REGION Network 36: UNIT 1 STATION 3 MEASURING RESET METHOD CONNECTION ALARM
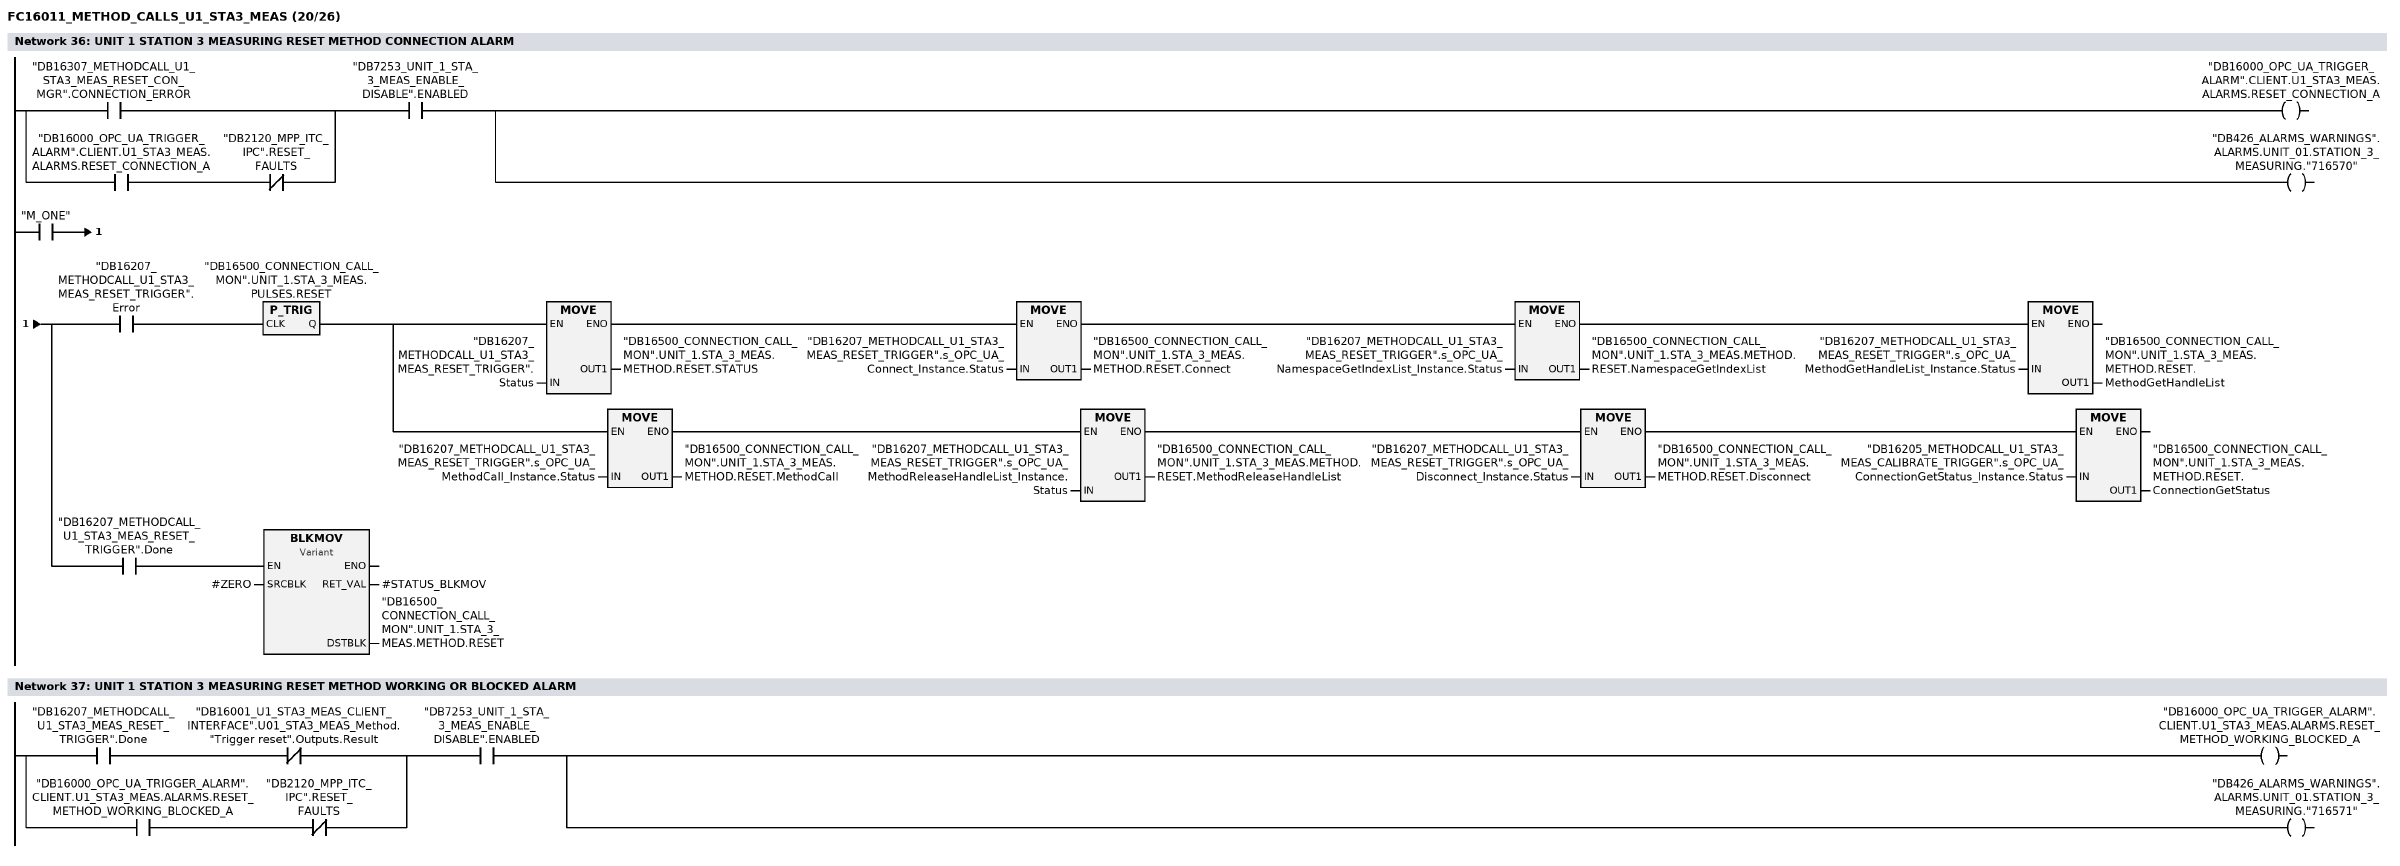
   RUNG wire#powerrail
      Contact( "DB16307_METHODCALL_U1_STA3_MEAS_RESET_CON_MGR".CONNECTION_ERROR )
      wire#w1
      Contact( "DB7253_UNIT_1_STA_3_MEAS_ENABLE_DISABLE".ENABLED )
      wire#w2
      Coil( "DB16000_OPC_UA_TRIGGER_ALARM".CLIENT.U1_STA3_MEAS.ALARMS.RESET_CONNECTION_A )
   END_RUNG
   RUNG wire#powerrail
      Contact( "DB16000_OPC_UA_TRIGGER_ALARM".CLIENT.U1_STA3_MEAS.ALARMS.RESET_CONNECTION_A )
      I_Contact( "DB2120_MPP_ITC_IPC".RESET_FAULTS )
   END_RUNG wire#w1
   RUNG wire#w2
      Coil( "DB426_ALARMS_WARNINGS".ALARMS.UNIT_01.STATION_3_MEASURING."716570" )
   END_RUNG
   RUNG wire#powerrail
      Contact( "M_ONE" )
      wire#w3
      Contact( "DB16207_METHODCALL_U1_STA3_MEAS_RESET_TRIGGER".Error )
      P_Trig( "DB16500_CONNECTION_CALL_MON".UNIT_1.STA_3_MEAS.PULSES.RESET )
      wire#w4
      Move(in := "DB16207_METHODCALL_U1_STA3_MEAS_RESET_TRIGGER".Status, out1 => "DB16500_CONNECTION_CALL_MON".UNIT_1.STA_3_MEAS.METHOD.RESET.STATUS)
      Move(in := "DB16207_METHODCALL_U1_STA3_MEAS_RESET_TRIGGER".s_OPC_UA_Connect_Instance.Status, out1 => "DB16500_CONNECTION_CALL_MON".UNIT_1.STA_3_MEAS.METHOD.RESET.Connect)
      Move(in := "DB16207_METHODCALL_U1_STA3_MEAS_RESET_TRIGGER".s_OPC_UA_NamespaceGetIndexList_Instance.Status, out1 => "DB16500_CONNECTION_CALL_MON".UNIT_1.STA_3_MEAS.METHOD.RESET.NamespaceGetIndexList)
      Move(in := "DB16207_METHODCALL_U1_STA3_MEAS_RESET_TRIGGER".s_OPC_UA_MethodGetHandleList_Instance.Status, out1 => "DB16500_CONNECTION_CALL_MON".UNIT_1.STA_3_MEAS.METHOD.RESET.MethodGetHandleList)
   END_RUNG
   RUNG wire#w4
      Move(in := "DB16207_METHODCALL_U1_STA3_MEAS_RESET_TRIGGER".s_OPC_UA_MethodCall_Instance.Status, out1 => "DB16500_CONNECTION_CALL_MON".UNIT_1.STA_3_MEAS.METHOD.RESET.MethodCall)
      Move(in := "DB16207_METHODCALL_U1_STA3_MEAS_RESET_TRIGGER".s_OPC_UA_MethodReleaseHandleList_Instance.Status, out1 => "DB16500_CONNECTION_CALL_MON".UNIT_1.STA_3_MEAS.METHOD.RESET.MethodReleaseHandleList)
      Move(in := "DB16207_METHODCALL_U1_STA3_MEAS_RESET_TRIGGER".s_OPC_UA_Disconnect_Instance.Status, out1 => "DB16500_CONNECTION_CALL_MON".UNIT_1.STA_3_MEAS.METHOD.RESET.Disconnect)
      Move(in := "DB16205_METHODCALL_U1_STA3_MEAS_CALIBRATE_TRIGGER".s_OPC_UA_ConnectionGetStatus_Instance.Status, out1 => "DB16500_CONNECTION_CALL_MON".UNIT_1.STA_3_MEAS.METHOD.RESET.ConnectionGetStatus)
   END_RUNG
   RUNG wire#w3
      Contact( "DB16207_METHODCALL_U1_STA3_MEAS_RESET_TRIGGER".Done )
      { S7_Templates := "blk_type := Variant" } BLKMOV(SRCBLK := #ZERO, RET_VAL => #STATUS_BLKMOV, DSTBLK => "DB16500_CONNECTION_CALL_MON".UNIT_1.STA_3_MEAS.METHOD.RESET)
   END_RUNG
   // the same network as SCL:
   "DB16000_OPC_UA_TRIGGER_ALARM".CLIENT.U1_STA3_MEAS.ALARMS.RESET_CONNECTION_A := ("DB16307_METHODCALL_U1_STA3_MEAS_RESET_CON_MGR".CONNECTION_ERROR OR ("DB16000_OPC_UA_TRIGGER_ALARM".CLIENT.U1_STA3_MEAS.ALARMS.RESET_CONNECTION_A AND NOT "DB2120_MPP_ITC_IPC".RESET_FAULTS)) AND "DB7253_UNIT_1_STA_3_MEAS_ENABLE_DISABLE".ENABLED;
   "DB426_ALARMS_WARNINGS".ALARMS.UNIT_01.STATION_3_MEASURING."716570" := "DB16000_OPC_UA_TRIGGER_ALARM".CLIENT.U1_STA3_MEAS.ALARMS.RESET_CONNECTION_A;
   #_w1 := "M_ONE" AND "DB16207_METHODCALL_U1_STA3_MEAS_RESET_TRIGGER".Error;
   #_w2 := #_w1 AND NOT "DB16500_CONNECTION_CALL_MON".UNIT_1.STA_3_MEAS.PULSES.RESET;   // rising edge
   "DB16500_CONNECTION_CALL_MON".UNIT_1.STA_3_MEAS.PULSES.RESET := #_w1;
   IF #_w2 THEN
       "DB16500_CONNECTION_CALL_MON".UNIT_1.STA_3_MEAS.METHOD.RESET.STATUS := "DB16207_METHODCALL_U1_STA3_MEAS_RESET_TRIGGER".Status;
       "DB16500_CONNECTION_CALL_MON".UNIT_1.STA_3_MEAS.METHOD.RESET.Connect := "DB16207_METHODCALL_U1_STA3_MEAS_RESET_TRIGGER".s_OPC_UA_Connect_Instance.Status;
       "DB16500_CONNECTION_CALL_MON".UNIT_1.STA_3_MEAS.METHOD.RESET.NamespaceGetIndexList := "DB16207_METHODCALL_U1_STA3_MEAS_RESET_TRIGGER".s_OPC_UA_NamespaceGetIndexList_Instance.Status;
       "DB16500_CONNECTION_CALL_MON".UNIT_1.STA_3_MEAS.METHOD.RESET.MethodGetHandleList := "DB16207_METHODCALL_U1_STA3_MEAS_RESET_TRIGGER".s_OPC_UA_MethodGetHandleList_Instance.Status;
       "DB16500_CONNECTION_CALL_MON".UNIT_1.STA_3_MEAS.METHOD.RESET.MethodCall := "DB16207_METHODCALL_U1_STA3_MEAS_RESET_TRIGGER".s_OPC_UA_MethodCall_Instance.Status;
       "DB16500_CONNECTION_CALL_MON".UNIT_1.STA_3_MEAS.METHOD.RESET.MethodReleaseHandleList := "DB16207_METHODCALL_U1_STA3_MEAS_RESET_TRIGGER".s_OPC_UA_MethodReleaseHandleList_Instance.Status;
       "DB16500_CONNECTION_CALL_MON".UNIT_1.STA_3_MEAS.METHOD.RESET.Disconnect := "DB16207_METHODCALL_U1_STA3_MEAS_RESET_TRIGGER".s_OPC_UA_Disconnect_Instance.Status;
       "DB16500_CONNECTION_CALL_MON".UNIT_1.STA_3_MEAS.METHOD.RESET.ConnectionGetStatus := "DB16205_METHODCALL_U1_STA3_MEAS_CALIBRATE_TRIGGER".s_OPC_UA_ConnectionGetStatus_Instance.Status;
   END_IF;
   IF "M_ONE" AND "DB16207_METHODCALL_U1_STA3_MEAS_RESET_TRIGGER".Done THEN
       #STATUS_BLKMOV := BLKMOV(SRCBLK := #ZERO,
                               DSTBLK => "DB16500_CONNECTION_CALL_MON".UNIT_1.STA_3_MEAS.METHOD.RESET);
   END_IF;
END_REGION

REGION Network 37: UNIT 1 STATION 3 MEASURING RESET METHOD WORKING OR BLOCKED ALARM
   RUNG wire#powerrail
      Contact( "DB16207_METHODCALL_U1_STA3_MEAS_RESET_TRIGGER".Done )
      I_Contact( "DB16001_U1_STA3_MEAS_CLIENT_INTERFACE".U01_STA3_MEAS_Method."Trigger reset".Outputs.Result )
      wire#w1
      Contact( "DB7253_UNIT_1_STA_3_MEAS_ENABLE_DISABLE".ENABLED )
      wire#w2
      Coil( "DB16000_OPC_UA_TRIGGER_ALARM".CLIENT.U1_STA3_MEAS.ALARMS.RESET_METHOD_WORKING_BLOCKED_A )
   END_RUNG
   RUNG wire#powerrail
      Contact( "DB16000_OPC_UA_TRIGGER_ALARM".CLIENT.U1_STA3_MEAS.ALARMS.RESET_METHOD_WORKING_BLOCKED_A )
      I_Contact( "DB2120_MPP_ITC_IPC".RESET_FAULTS )
   END_RUNG wire#w1
   RUNG wire#w2
      Coil( "DB426_ALARMS_WARNINGS".ALARMS.UNIT_01.STATION_3_MEASURING."716571" )
   END_RUNG
   // the same network as SCL:
   "DB16000_OPC_UA_TRIGGER_ALARM".CLIENT.U1_STA3_MEAS.ALARMS.RESET_METHOD_WORKING_BLOCKED_A := (("DB16207_METHODCALL_U1_STA3_MEAS_RESET_TRIGGER".Done AND NOT "DB16001_U1_STA3_MEAS_CLIENT_INTERFACE".U01_STA3_MEAS_Method."Trigger reset".Outputs.Result) OR ("DB16000_OPC_UA_TRIGGER_ALARM".CLIENT.U1_STA3_MEAS.ALARMS.RESET_METHOD_WORKING_BLOCKED_A AND NOT "DB2120_MPP_ITC_IPC".RESET_FAULTS)) AND "DB7253_UNIT_1_STA_3_MEAS_ENABLE_DISABLE".ENABLED;
   "DB426_ALARMS_WARNINGS".ALARMS.UNIT_01.STATION_3_MEASURING."716571" := "DB16000_OPC_UA_TRIGGER_ALARM".CLIENT.U1_STA3_MEAS.ALARMS.RESET_METHOD_WORKING_BLOCKED_A;
END_REGION

REGION Network 38: UNIT 1 STATION 3 MEASURING READ VARIABLES CONNECTION ALARM
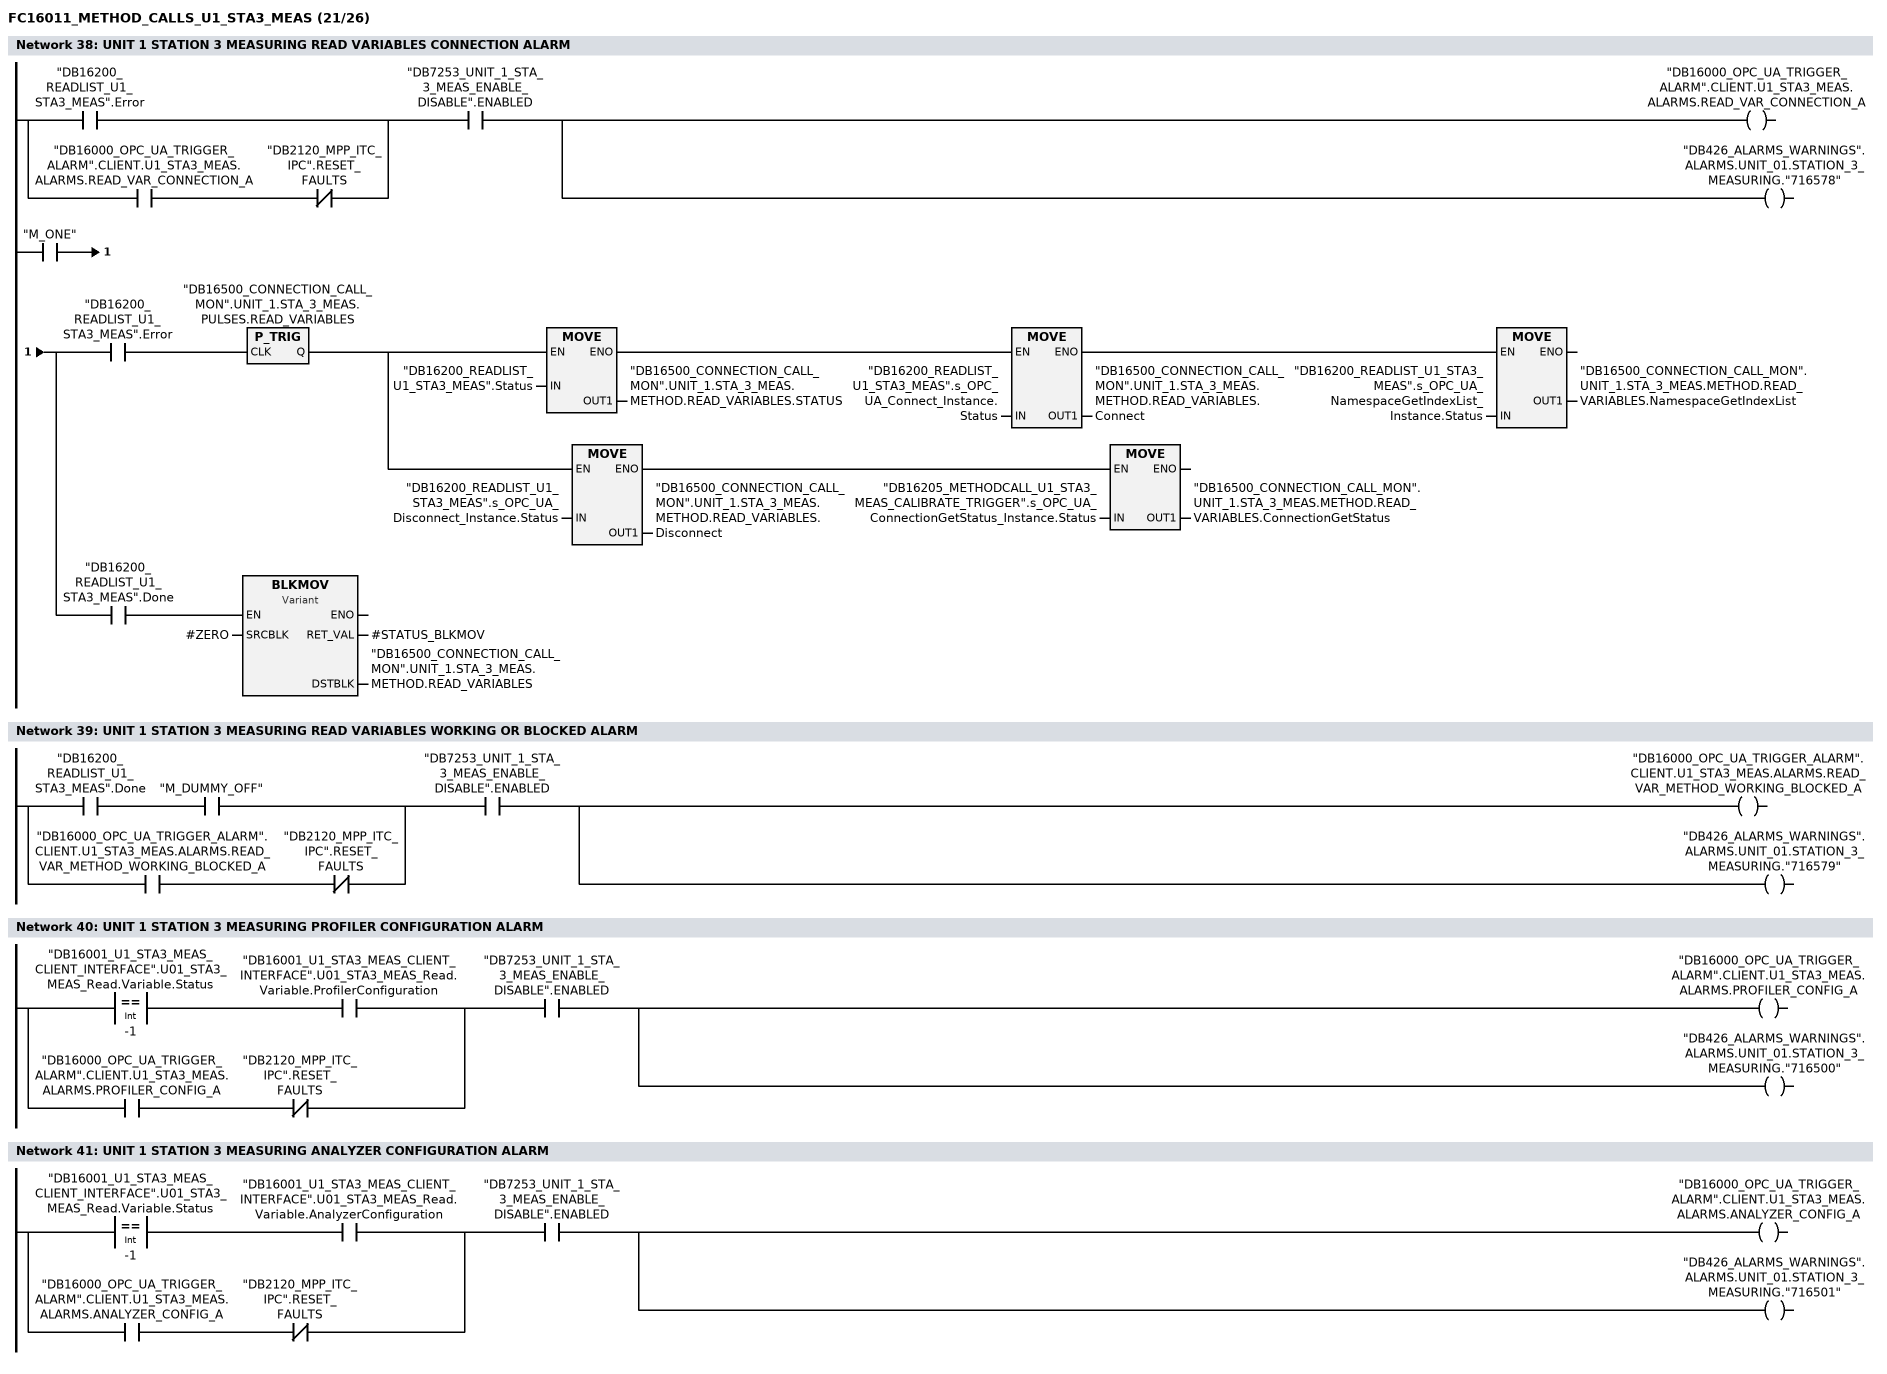
   RUNG wire#powerrail
      Contact( "DB16200_READLIST_U1_STA3_MEAS".Error )
      wire#w1
      Contact( "DB7253_UNIT_1_STA_3_MEAS_ENABLE_DISABLE".ENABLED )
      wire#w2
      Coil( "DB16000_OPC_UA_TRIGGER_ALARM".CLIENT.U1_STA3_MEAS.ALARMS.READ_VAR_CONNECTION_A )
   END_RUNG
   RUNG wire#powerrail
      Contact( "DB16000_OPC_UA_TRIGGER_ALARM".CLIENT.U1_STA3_MEAS.ALARMS.READ_VAR_CONNECTION_A )
      I_Contact( "DB2120_MPP_ITC_IPC".RESET_FAULTS )
   END_RUNG wire#w1
   RUNG wire#w2
      Coil( "DB426_ALARMS_WARNINGS".ALARMS.UNIT_01.STATION_3_MEASURING."716578" )
   END_RUNG
   RUNG wire#powerrail
      Contact( "M_ONE" )
      wire#w3
      Contact( "DB16200_READLIST_U1_STA3_MEAS".Error )
      P_Trig( "DB16500_CONNECTION_CALL_MON".UNIT_1.STA_3_MEAS.PULSES.READ_VARIABLES )
      wire#w4
      Move(in := "DB16200_READLIST_U1_STA3_MEAS".Status, out1 => "DB16500_CONNECTION_CALL_MON".UNIT_1.STA_3_MEAS.METHOD.READ_VARIABLES.STATUS)
      Move(in := "DB16200_READLIST_U1_STA3_MEAS".s_OPC_UA_Connect_Instance.Status, out1 => "DB16500_CONNECTION_CALL_MON".UNIT_1.STA_3_MEAS.METHOD.READ_VARIABLES.Connect)
      Move(in := "DB16200_READLIST_U1_STA3_MEAS".s_OPC_UA_NamespaceGetIndexList_Instance.Status, out1 => "DB16500_CONNECTION_CALL_MON".UNIT_1.STA_3_MEAS.METHOD.READ_VARIABLES.NamespaceGetIndexList)
   END_RUNG
   RUNG wire#w4
      Move(in := "DB16200_READLIST_U1_STA3_MEAS".s_OPC_UA_Disconnect_Instance.Status, out1 => "DB16500_CONNECTION_CALL_MON".UNIT_1.STA_3_MEAS.METHOD.READ_VARIABLES.Disconnect)
      Move(in := "DB16205_METHODCALL_U1_STA3_MEAS_CALIBRATE_TRIGGER".s_OPC_UA_ConnectionGetStatus_Instance.Status, out1 => "DB16500_CONNECTION_CALL_MON".UNIT_1.STA_3_MEAS.METHOD.READ_VARIABLES.ConnectionGetStatus)
   END_RUNG
   RUNG wire#w3
      Contact( "DB16200_READLIST_U1_STA3_MEAS".Done )
      { S7_Templates := "blk_type := Variant" } BLKMOV(SRCBLK := #ZERO, RET_VAL => #STATUS_BLKMOV, DSTBLK => "DB16500_CONNECTION_CALL_MON".UNIT_1.STA_3_MEAS.METHOD.READ_VARIABLES)
   END_RUNG
   // the same network as SCL:
   "DB16000_OPC_UA_TRIGGER_ALARM".CLIENT.U1_STA3_MEAS.ALARMS.READ_VAR_CONNECTION_A := ("DB16200_READLIST_U1_STA3_MEAS".Error OR ("DB16000_OPC_UA_TRIGGER_ALARM".CLIENT.U1_STA3_MEAS.ALARMS.READ_VAR_CONNECTION_A AND NOT "DB2120_MPP_ITC_IPC".RESET_FAULTS)) AND "DB7253_UNIT_1_STA_3_MEAS_ENABLE_DISABLE".ENABLED;
   "DB426_ALARMS_WARNINGS".ALARMS.UNIT_01.STATION_3_MEASURING."716578" := "DB16000_OPC_UA_TRIGGER_ALARM".CLIENT.U1_STA3_MEAS.ALARMS.READ_VAR_CONNECTION_A;
   #_w1 := "M_ONE" AND "DB16200_READLIST_U1_STA3_MEAS".Error;
   #_w2 := #_w1 AND NOT "DB16500_CONNECTION_CALL_MON".UNIT_1.STA_3_MEAS.PULSES.READ_VARIABLES;   // rising edge
   "DB16500_CONNECTION_CALL_MON".UNIT_1.STA_3_MEAS.PULSES.READ_VARIABLES := #_w1;
   IF #_w2 THEN
       "DB16500_CONNECTION_CALL_MON".UNIT_1.STA_3_MEAS.METHOD.READ_VARIABLES.STATUS := "DB16200_READLIST_U1_STA3_MEAS".Status;
       "DB16500_CONNECTION_CALL_MON".UNIT_1.STA_3_MEAS.METHOD.READ_VARIABLES.Connect := "DB16200_READLIST_U1_STA3_MEAS".s_OPC_UA_Connect_Instance.Status;
       "DB16500_CONNECTION_CALL_MON".UNIT_1.STA_3_MEAS.METHOD.READ_VARIABLES.NamespaceGetIndexList := "DB16200_READLIST_U1_STA3_MEAS".s_OPC_UA_NamespaceGetIndexList_Instance.Status;
       "DB16500_CONNECTION_CALL_MON".UNIT_1.STA_3_MEAS.METHOD.READ_VARIABLES.Disconnect := "DB16200_READLIST_U1_STA3_MEAS".s_OPC_UA_Disconnect_Instance.Status;
       "DB16500_CONNECTION_CALL_MON".UNIT_1.STA_3_MEAS.METHOD.READ_VARIABLES.ConnectionGetStatus := "DB16205_METHODCALL_U1_STA3_MEAS_CALIBRATE_TRIGGER".s_OPC_UA_ConnectionGetStatus_Instance.Status;
   END_IF;
   IF "M_ONE" AND "DB16200_READLIST_U1_STA3_MEAS".Done THEN
       #STATUS_BLKMOV := BLKMOV(SRCBLK := #ZERO,
                               DSTBLK => "DB16500_CONNECTION_CALL_MON".UNIT_1.STA_3_MEAS.METHOD.READ_VARIABLES);
   END_IF;
END_REGION

REGION Network 39: UNIT 1 STATION 3 MEASURING READ VARIABLES WORKING OR BLOCKED ALARM
   RUNG wire#powerrail
      Contact( "DB16200_READLIST_U1_STA3_MEAS".Done )
      Contact( "M_DUMMY_OFF" )
      wire#w1
      Contact( "DB7253_UNIT_1_STA_3_MEAS_ENABLE_DISABLE".ENABLED )
      wire#w2
      Coil( "DB16000_OPC_UA_TRIGGER_ALARM".CLIENT.U1_STA3_MEAS.ALARMS.READ_VAR_METHOD_WORKING_BLOCKED_A )
   END_RUNG
   RUNG wire#powerrail
      Contact( "DB16000_OPC_UA_TRIGGER_ALARM".CLIENT.U1_STA3_MEAS.ALARMS.READ_VAR_METHOD_WORKING_BLOCKED_A )
      I_Contact( "DB2120_MPP_ITC_IPC".RESET_FAULTS )
   END_RUNG wire#w1
   RUNG wire#w2
      Coil( "DB426_ALARMS_WARNINGS".ALARMS.UNIT_01.STATION_3_MEASURING."716579" )
   END_RUNG
   // the same network as SCL:
   "DB16000_OPC_UA_TRIGGER_ALARM".CLIENT.U1_STA3_MEAS.ALARMS.READ_VAR_METHOD_WORKING_BLOCKED_A := (("DB16200_READLIST_U1_STA3_MEAS".Done AND "M_DUMMY_OFF") OR ("DB16000_OPC_UA_TRIGGER_ALARM".CLIENT.U1_STA3_MEAS.ALARMS.READ_VAR_METHOD_WORKING_BLOCKED_A AND NOT "DB2120_MPP_ITC_IPC".RESET_FAULTS)) AND "DB7253_UNIT_1_STA_3_MEAS_ENABLE_DISABLE".ENABLED;
   "DB426_ALARMS_WARNINGS".ALARMS.UNIT_01.STATION_3_MEASURING."716579" := "DB16000_OPC_UA_TRIGGER_ALARM".CLIENT.U1_STA3_MEAS.ALARMS.READ_VAR_METHOD_WORKING_BLOCKED_A;
END_REGION

REGION Network 40: UNIT 1 STATION 3 MEASURING PROFILER CONFIGURATION ALARM
   RUNG wire#powerrail
      { S7_Templates := "SrcType := Int" } EQ_Contact(in1 := "DB16001_U1_STA3_MEAS_CLIENT_INTERFACE".U01_STA3_MEAS_Read.Variable.Status, in2 := -1)
      Contact( "DB16001_U1_STA3_MEAS_CLIENT_INTERFACE".U01_STA3_MEAS_Read.Variable.ProfilerConfiguration )
      wire#w1
      Contact( "DB7253_UNIT_1_STA_3_MEAS_ENABLE_DISABLE".ENABLED )
      wire#w2
      Coil( "DB16000_OPC_UA_TRIGGER_ALARM".CLIENT.U1_STA3_MEAS.ALARMS.PROFILER_CONFIG_A )
   END_RUNG
   RUNG wire#powerrail
      Contact( "DB16000_OPC_UA_TRIGGER_ALARM".CLIENT.U1_STA3_MEAS.ALARMS.PROFILER_CONFIG_A )
      I_Contact( "DB2120_MPP_ITC_IPC".RESET_FAULTS )
   END_RUNG wire#w1
   RUNG wire#w2
      Coil( "DB426_ALARMS_WARNINGS".ALARMS.UNIT_01.STATION_3_MEASURING."716500" )
   END_RUNG
   // the same network as SCL:
   "DB16000_OPC_UA_TRIGGER_ALARM".CLIENT.U1_STA3_MEAS.ALARMS.PROFILER_CONFIG_A := ((("DB16001_U1_STA3_MEAS_CLIENT_INTERFACE".U01_STA3_MEAS_Read.Variable.Status = (-1)) AND "DB16001_U1_STA3_MEAS_CLIENT_INTERFACE".U01_STA3_MEAS_Read.Variable.ProfilerConfiguration) OR ("DB16000_OPC_UA_TRIGGER_ALARM".CLIENT.U1_STA3_MEAS.ALARMS.PROFILER_CONFIG_A AND NOT "DB2120_MPP_ITC_IPC".RESET_FAULTS)) AND "DB7253_UNIT_1_STA_3_MEAS_ENABLE_DISABLE".ENABLED;
   "DB426_ALARMS_WARNINGS".ALARMS.UNIT_01.STATION_3_MEASURING."716500" := "DB16000_OPC_UA_TRIGGER_ALARM".CLIENT.U1_STA3_MEAS.ALARMS.PROFILER_CONFIG_A;
END_REGION

REGION Network 41: UNIT 1 STATION 3 MEASURING ANALYZER CONFIGURATION ALARM
   RUNG wire#powerrail
      { S7_Templates := "SrcType := Int" } EQ_Contact(in1 := "DB16001_U1_STA3_MEAS_CLIENT_INTERFACE".U01_STA3_MEAS_Read.Variable.Status, in2 := -1)
      Contact( "DB16001_U1_STA3_MEAS_CLIENT_INTERFACE".U01_STA3_MEAS_Read.Variable.AnalyzerConfiguration )
      wire#w1
      Contact( "DB7253_UNIT_1_STA_3_MEAS_ENABLE_DISABLE".ENABLED )
      wire#w2
      Coil( "DB16000_OPC_UA_TRIGGER_ALARM".CLIENT.U1_STA3_MEAS.ALARMS.ANALYZER_CONFIG_A )
   END_RUNG
   RUNG wire#powerrail
      Contact( "DB16000_OPC_UA_TRIGGER_ALARM".CLIENT.U1_STA3_MEAS.ALARMS.ANALYZER_CONFIG_A )
      I_Contact( "DB2120_MPP_ITC_IPC".RESET_FAULTS )
   END_RUNG wire#w1
   RUNG wire#w2
      Coil( "DB426_ALARMS_WARNINGS".ALARMS.UNIT_01.STATION_3_MEASURING."716501" )
   END_RUNG
   // the same network as SCL:
   "DB16000_OPC_UA_TRIGGER_ALARM".CLIENT.U1_STA3_MEAS.ALARMS.ANALYZER_CONFIG_A := ((("DB16001_U1_STA3_MEAS_CLIENT_INTERFACE".U01_STA3_MEAS_Read.Variable.Status = (-1)) AND "DB16001_U1_STA3_MEAS_CLIENT_INTERFACE".U01_STA3_MEAS_Read.Variable.AnalyzerConfiguration) OR ("DB16000_OPC_UA_TRIGGER_ALARM".CLIENT.U1_STA3_MEAS.ALARMS.ANALYZER_CONFIG_A AND NOT "DB2120_MPP_ITC_IPC".RESET_FAULTS)) AND "DB7253_UNIT_1_STA_3_MEAS_ENABLE_DISABLE".ENABLED;
   "DB426_ALARMS_WARNINGS".ALARMS.UNIT_01.STATION_3_MEASURING."716501" := "DB16000_OPC_UA_TRIGGER_ALARM".CLIENT.U1_STA3_MEAS.ALARMS.ANALYZER_CONFIG_A;
END_REGION

REGION Network 42: UNIT 1 STATION 3 MEASURING DMC STRUCTURE ALARM
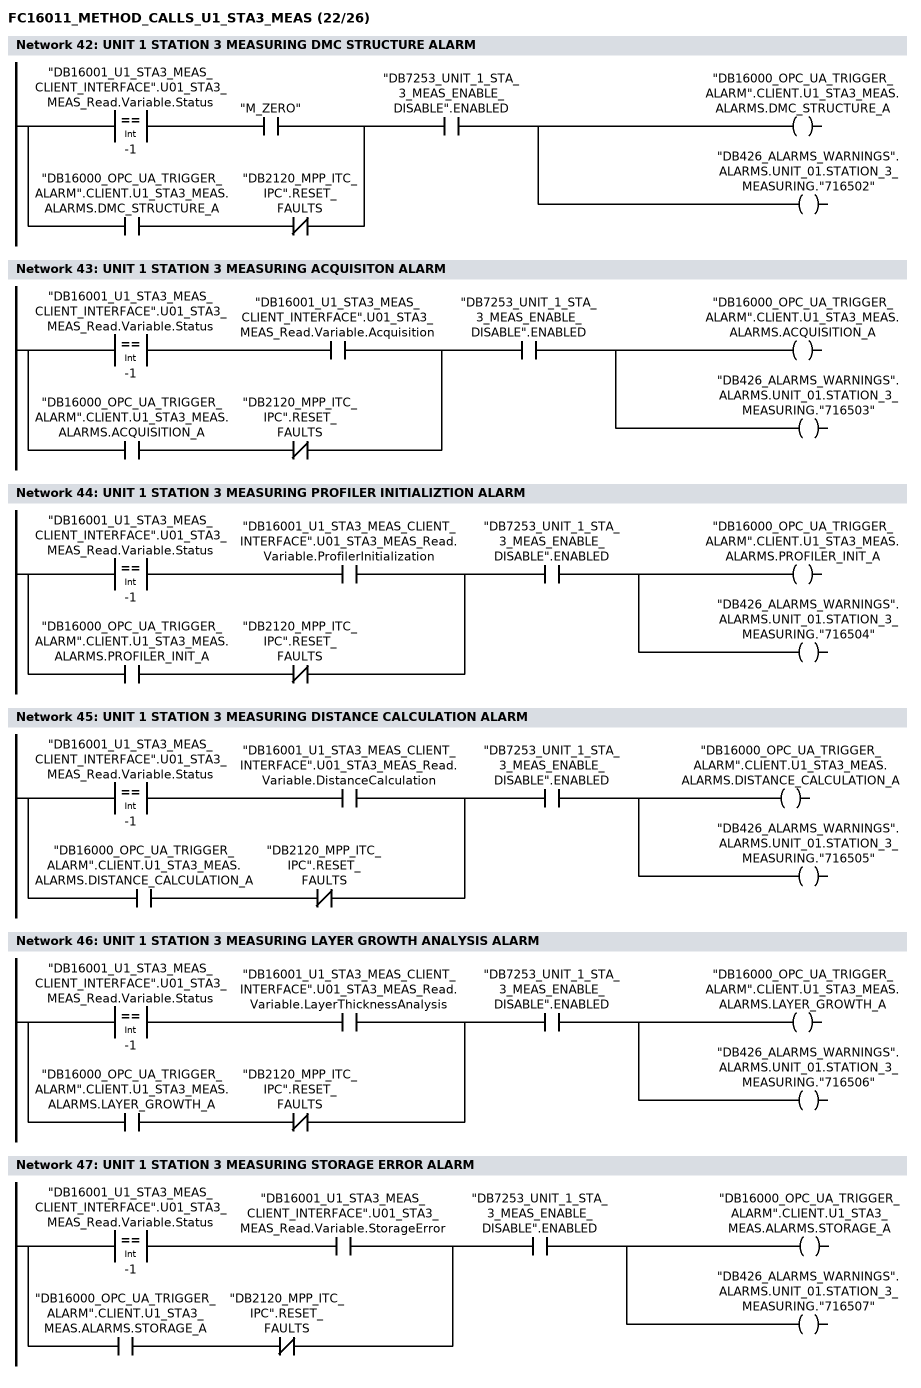
   RUNG wire#powerrail
      { S7_Templates := "SrcType := Int" } EQ_Contact(in1 := "DB16001_U1_STA3_MEAS_CLIENT_INTERFACE".U01_STA3_MEAS_Read.Variable.Status, in2 := -1)
      Contact( "M_ZERO" )
      wire#w1
      Contact( "DB7253_UNIT_1_STA_3_MEAS_ENABLE_DISABLE".ENABLED )
      wire#w2
      Coil( "DB16000_OPC_UA_TRIGGER_ALARM".CLIENT.U1_STA3_MEAS.ALARMS.DMC_STRUCTURE_A )
   END_RUNG
   RUNG wire#powerrail
      Contact( "DB16000_OPC_UA_TRIGGER_ALARM".CLIENT.U1_STA3_MEAS.ALARMS.DMC_STRUCTURE_A )
      I_Contact( "DB2120_MPP_ITC_IPC".RESET_FAULTS )
   END_RUNG wire#w1
   RUNG wire#w2
      Coil( "DB426_ALARMS_WARNINGS".ALARMS.UNIT_01.STATION_3_MEASURING."716502" )
   END_RUNG
   // the same network as SCL:
   "DB16000_OPC_UA_TRIGGER_ALARM".CLIENT.U1_STA3_MEAS.ALARMS.DMC_STRUCTURE_A := ((("DB16001_U1_STA3_MEAS_CLIENT_INTERFACE".U01_STA3_MEAS_Read.Variable.Status = (-1)) AND "M_ZERO") OR ("DB16000_OPC_UA_TRIGGER_ALARM".CLIENT.U1_STA3_MEAS.ALARMS.DMC_STRUCTURE_A AND NOT "DB2120_MPP_ITC_IPC".RESET_FAULTS)) AND "DB7253_UNIT_1_STA_3_MEAS_ENABLE_DISABLE".ENABLED;
   "DB426_ALARMS_WARNINGS".ALARMS.UNIT_01.STATION_3_MEASURING."716502" := "DB16000_OPC_UA_TRIGGER_ALARM".CLIENT.U1_STA3_MEAS.ALARMS.DMC_STRUCTURE_A;
END_REGION

REGION Network 43: UNIT 1 STATION 3 MEASURING ACQUISITON ALARM
   RUNG wire#powerrail
      { S7_Templates := "SrcType := Int" } EQ_Contact(in1 := "DB16001_U1_STA3_MEAS_CLIENT_INTERFACE".U01_STA3_MEAS_Read.Variable.Status, in2 := -1)
      Contact( "DB16001_U1_STA3_MEAS_CLIENT_INTERFACE".U01_STA3_MEAS_Read.Variable.Acquisition )
      wire#w1
      Contact( "DB7253_UNIT_1_STA_3_MEAS_ENABLE_DISABLE".ENABLED )
      wire#w2
      Coil( "DB16000_OPC_UA_TRIGGER_ALARM".CLIENT.U1_STA3_MEAS.ALARMS.ACQUISITION_A )
   END_RUNG
   RUNG wire#powerrail
      Contact( "DB16000_OPC_UA_TRIGGER_ALARM".CLIENT.U1_STA3_MEAS.ALARMS.ACQUISITION_A )
      I_Contact( "DB2120_MPP_ITC_IPC".RESET_FAULTS )
   END_RUNG wire#w1
   RUNG wire#w2
      Coil( "DB426_ALARMS_WARNINGS".ALARMS.UNIT_01.STATION_3_MEASURING."716503" )
   END_RUNG
   // the same network as SCL:
   "DB16000_OPC_UA_TRIGGER_ALARM".CLIENT.U1_STA3_MEAS.ALARMS.ACQUISITION_A := ((("DB16001_U1_STA3_MEAS_CLIENT_INTERFACE".U01_STA3_MEAS_Read.Variable.Status = (-1)) AND "DB16001_U1_STA3_MEAS_CLIENT_INTERFACE".U01_STA3_MEAS_Read.Variable.Acquisition) OR ("DB16000_OPC_UA_TRIGGER_ALARM".CLIENT.U1_STA3_MEAS.ALARMS.ACQUISITION_A AND NOT "DB2120_MPP_ITC_IPC".RESET_FAULTS)) AND "DB7253_UNIT_1_STA_3_MEAS_ENABLE_DISABLE".ENABLED;
   "DB426_ALARMS_WARNINGS".ALARMS.UNIT_01.STATION_3_MEASURING."716503" := "DB16000_OPC_UA_TRIGGER_ALARM".CLIENT.U1_STA3_MEAS.ALARMS.ACQUISITION_A;
END_REGION

REGION Network 44: UNIT 1 STATION 3 MEASURING PROFILER INITIALIZTION ALARM
   RUNG wire#powerrail
      { S7_Templates := "SrcType := Int" } EQ_Contact(in1 := "DB16001_U1_STA3_MEAS_CLIENT_INTERFACE".U01_STA3_MEAS_Read.Variable.Status, in2 := -1)
      Contact( "DB16001_U1_STA3_MEAS_CLIENT_INTERFACE".U01_STA3_MEAS_Read.Variable.ProfilerInitialization )
      wire#w1
      Contact( "DB7253_UNIT_1_STA_3_MEAS_ENABLE_DISABLE".ENABLED )
      wire#w2
      Coil( "DB16000_OPC_UA_TRIGGER_ALARM".CLIENT.U1_STA3_MEAS.ALARMS.PROFILER_INIT_A )
   END_RUNG
   RUNG wire#powerrail
      Contact( "DB16000_OPC_UA_TRIGGER_ALARM".CLIENT.U1_STA3_MEAS.ALARMS.PROFILER_INIT_A )
      I_Contact( "DB2120_MPP_ITC_IPC".RESET_FAULTS )
   END_RUNG wire#w1
   RUNG wire#w2
      Coil( "DB426_ALARMS_WARNINGS".ALARMS.UNIT_01.STATION_3_MEASURING."716504" )
   END_RUNG
   // the same network as SCL:
   "DB16000_OPC_UA_TRIGGER_ALARM".CLIENT.U1_STA3_MEAS.ALARMS.PROFILER_INIT_A := ((("DB16001_U1_STA3_MEAS_CLIENT_INTERFACE".U01_STA3_MEAS_Read.Variable.Status = (-1)) AND "DB16001_U1_STA3_MEAS_CLIENT_INTERFACE".U01_STA3_MEAS_Read.Variable.ProfilerInitialization) OR ("DB16000_OPC_UA_TRIGGER_ALARM".CLIENT.U1_STA3_MEAS.ALARMS.PROFILER_INIT_A AND NOT "DB2120_MPP_ITC_IPC".RESET_FAULTS)) AND "DB7253_UNIT_1_STA_3_MEAS_ENABLE_DISABLE".ENABLED;
   "DB426_ALARMS_WARNINGS".ALARMS.UNIT_01.STATION_3_MEASURING."716504" := "DB16000_OPC_UA_TRIGGER_ALARM".CLIENT.U1_STA3_MEAS.ALARMS.PROFILER_INIT_A;
END_REGION

REGION Network 45: UNIT 1 STATION 3 MEASURING DISTANCE CALCULATION ALARM
   RUNG wire#powerrail
      { S7_Templates := "SrcType := Int" } EQ_Contact(in1 := "DB16001_U1_STA3_MEAS_CLIENT_INTERFACE".U01_STA3_MEAS_Read.Variable.Status, in2 := -1)
      Contact( "DB16001_U1_STA3_MEAS_CLIENT_INTERFACE".U01_STA3_MEAS_Read.Variable.DistanceCalculation )
      wire#w1
      Contact( "DB7253_UNIT_1_STA_3_MEAS_ENABLE_DISABLE".ENABLED )
      wire#w2
      Coil( "DB16000_OPC_UA_TRIGGER_ALARM".CLIENT.U1_STA3_MEAS.ALARMS.DISTANCE_CALCULATION_A )
   END_RUNG
   RUNG wire#powerrail
      Contact( "DB16000_OPC_UA_TRIGGER_ALARM".CLIENT.U1_STA3_MEAS.ALARMS.DISTANCE_CALCULATION_A )
      I_Contact( "DB2120_MPP_ITC_IPC".RESET_FAULTS )
   END_RUNG wire#w1
   RUNG wire#w2
      Coil( "DB426_ALARMS_WARNINGS".ALARMS.UNIT_01.STATION_3_MEASURING."716505" )
   END_RUNG
   // the same network as SCL:
   "DB16000_OPC_UA_TRIGGER_ALARM".CLIENT.U1_STA3_MEAS.ALARMS.DISTANCE_CALCULATION_A := ((("DB16001_U1_STA3_MEAS_CLIENT_INTERFACE".U01_STA3_MEAS_Read.Variable.Status = (-1)) AND "DB16001_U1_STA3_MEAS_CLIENT_INTERFACE".U01_STA3_MEAS_Read.Variable.DistanceCalculation) OR ("DB16000_OPC_UA_TRIGGER_ALARM".CLIENT.U1_STA3_MEAS.ALARMS.DISTANCE_CALCULATION_A AND NOT "DB2120_MPP_ITC_IPC".RESET_FAULTS)) AND "DB7253_UNIT_1_STA_3_MEAS_ENABLE_DISABLE".ENABLED;
   "DB426_ALARMS_WARNINGS".ALARMS.UNIT_01.STATION_3_MEASURING."716505" := "DB16000_OPC_UA_TRIGGER_ALARM".CLIENT.U1_STA3_MEAS.ALARMS.DISTANCE_CALCULATION_A;
END_REGION

REGION Network 46: UNIT 1 STATION 3 MEASURING LAYER GROWTH ANALYSIS ALARM
   RUNG wire#powerrail
      { S7_Templates := "SrcType := Int" } EQ_Contact(in1 := "DB16001_U1_STA3_MEAS_CLIENT_INTERFACE".U01_STA3_MEAS_Read.Variable.Status, in2 := -1)
      Contact( "DB16001_U1_STA3_MEAS_CLIENT_INTERFACE".U01_STA3_MEAS_Read.Variable.LayerThicknessAnalysis )
      wire#w1
      Contact( "DB7253_UNIT_1_STA_3_MEAS_ENABLE_DISABLE".ENABLED )
      wire#w2
      Coil( "DB16000_OPC_UA_TRIGGER_ALARM".CLIENT.U1_STA3_MEAS.ALARMS.LAYER_GROWTH_A )
   END_RUNG
   RUNG wire#powerrail
      Contact( "DB16000_OPC_UA_TRIGGER_ALARM".CLIENT.U1_STA3_MEAS.ALARMS.LAYER_GROWTH_A )
      I_Contact( "DB2120_MPP_ITC_IPC".RESET_FAULTS )
   END_RUNG wire#w1
   RUNG wire#w2
      Coil( "DB426_ALARMS_WARNINGS".ALARMS.UNIT_01.STATION_3_MEASURING."716506" )
   END_RUNG
   // the same network as SCL:
   "DB16000_OPC_UA_TRIGGER_ALARM".CLIENT.U1_STA3_MEAS.ALARMS.LAYER_GROWTH_A := ((("DB16001_U1_STA3_MEAS_CLIENT_INTERFACE".U01_STA3_MEAS_Read.Variable.Status = (-1)) AND "DB16001_U1_STA3_MEAS_CLIENT_INTERFACE".U01_STA3_MEAS_Read.Variable.LayerThicknessAnalysis) OR ("DB16000_OPC_UA_TRIGGER_ALARM".CLIENT.U1_STA3_MEAS.ALARMS.LAYER_GROWTH_A AND NOT "DB2120_MPP_ITC_IPC".RESET_FAULTS)) AND "DB7253_UNIT_1_STA_3_MEAS_ENABLE_DISABLE".ENABLED;
   "DB426_ALARMS_WARNINGS".ALARMS.UNIT_01.STATION_3_MEASURING."716506" := "DB16000_OPC_UA_TRIGGER_ALARM".CLIENT.U1_STA3_MEAS.ALARMS.LAYER_GROWTH_A;
END_REGION

REGION Network 47: UNIT 1 STATION 3 MEASURING STORAGE ERROR ALARM
   RUNG wire#powerrail
      { S7_Templates := "SrcType := Int" } EQ_Contact(in1 := "DB16001_U1_STA3_MEAS_CLIENT_INTERFACE".U01_STA3_MEAS_Read.Variable.Status, in2 := -1)
      Contact( "DB16001_U1_STA3_MEAS_CLIENT_INTERFACE".U01_STA3_MEAS_Read.Variable.StorageError )
      wire#w1
      Contact( "DB7253_UNIT_1_STA_3_MEAS_ENABLE_DISABLE".ENABLED )
      wire#w2
      Coil( "DB16000_OPC_UA_TRIGGER_ALARM".CLIENT.U1_STA3_MEAS.ALARMS.STORAGE_A )
   END_RUNG
   RUNG wire#powerrail
      Contact( "DB16000_OPC_UA_TRIGGER_ALARM".CLIENT.U1_STA3_MEAS.ALARMS.STORAGE_A )
      I_Contact( "DB2120_MPP_ITC_IPC".RESET_FAULTS )
   END_RUNG wire#w1
   RUNG wire#w2
      Coil( "DB426_ALARMS_WARNINGS".ALARMS.UNIT_01.STATION_3_MEASURING."716507" )
   END_RUNG
   // the same network as SCL:
   "DB16000_OPC_UA_TRIGGER_ALARM".CLIENT.U1_STA3_MEAS.ALARMS.STORAGE_A := ((("DB16001_U1_STA3_MEAS_CLIENT_INTERFACE".U01_STA3_MEAS_Read.Variable.Status = (-1)) AND "DB16001_U1_STA3_MEAS_CLIENT_INTERFACE".U01_STA3_MEAS_Read.Variable.StorageError) OR ("DB16000_OPC_UA_TRIGGER_ALARM".CLIENT.U1_STA3_MEAS.ALARMS.STORAGE_A AND NOT "DB2120_MPP_ITC_IPC".RESET_FAULTS)) AND "DB7253_UNIT_1_STA_3_MEAS_ENABLE_DISABLE".ENABLED;
   "DB426_ALARMS_WARNINGS".ALARMS.UNIT_01.STATION_3_MEASURING."716507" := "DB16000_OPC_UA_TRIGGER_ALARM".CLIENT.U1_STA3_MEAS.ALARMS.STORAGE_A;
END_REGION

REGION Network 48: UNIT 1 STATION 3 MEASURING DATABASE CONNECTION ALARM
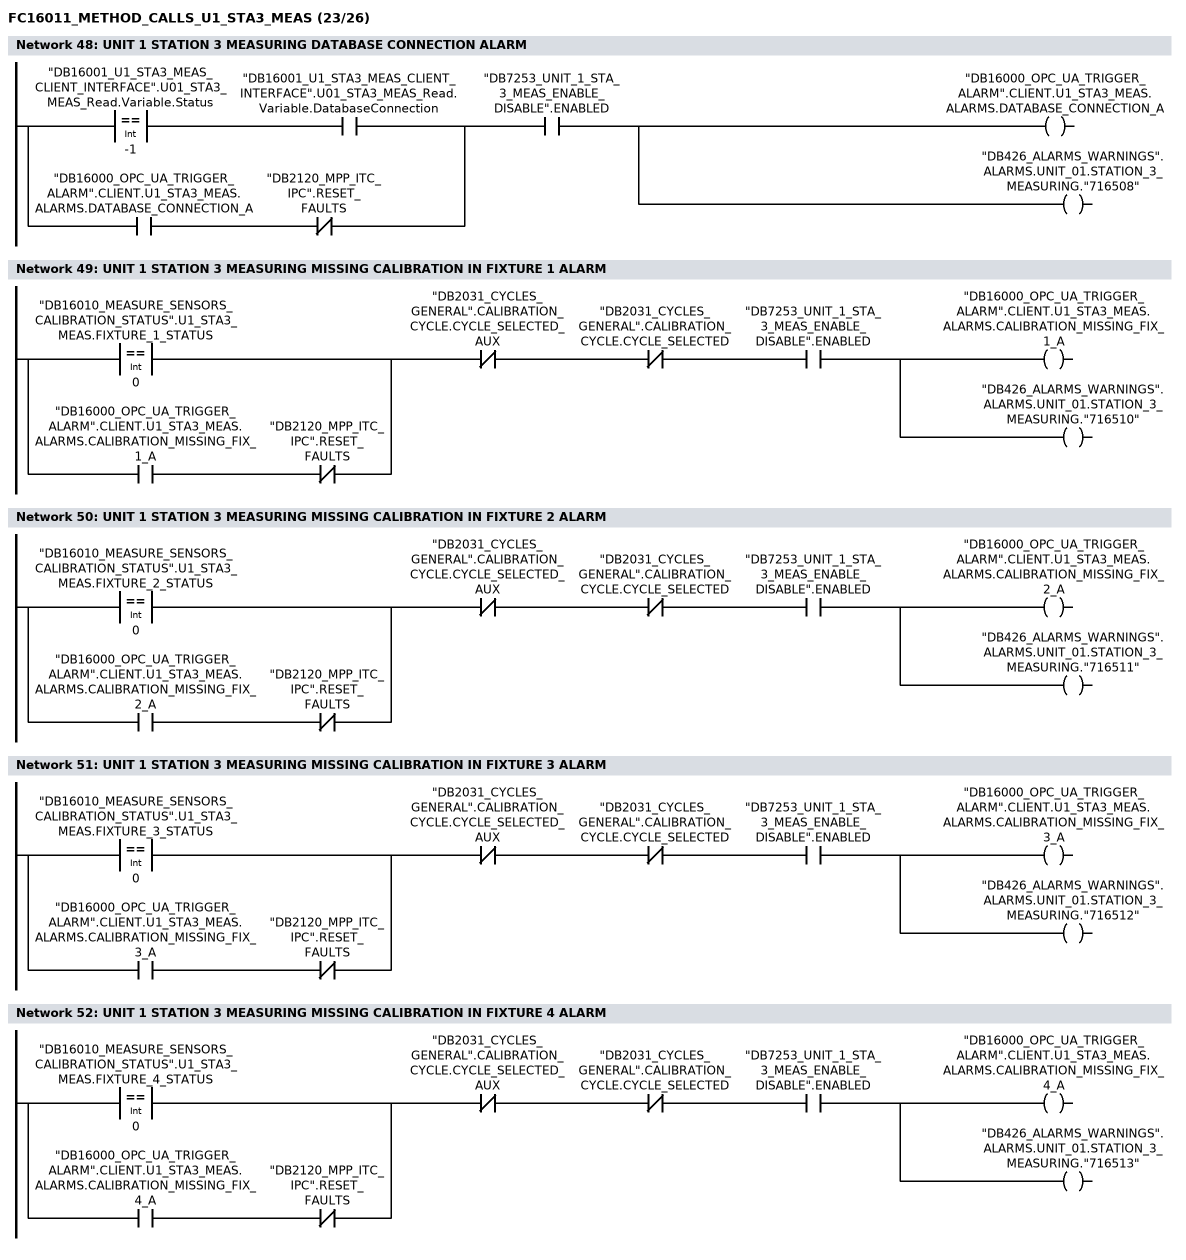
   RUNG wire#powerrail
      { S7_Templates := "SrcType := Int" } EQ_Contact(in1 := "DB16001_U1_STA3_MEAS_CLIENT_INTERFACE".U01_STA3_MEAS_Read.Variable.Status, in2 := -1)
      Contact( "DB16001_U1_STA3_MEAS_CLIENT_INTERFACE".U01_STA3_MEAS_Read.Variable.DatabaseConnection )
      wire#w1
      Contact( "DB7253_UNIT_1_STA_3_MEAS_ENABLE_DISABLE".ENABLED )
      wire#w2
      Coil( "DB16000_OPC_UA_TRIGGER_ALARM".CLIENT.U1_STA3_MEAS.ALARMS.DATABASE_CONNECTION_A )
   END_RUNG
   RUNG wire#powerrail
      Contact( "DB16000_OPC_UA_TRIGGER_ALARM".CLIENT.U1_STA3_MEAS.ALARMS.DATABASE_CONNECTION_A )
      I_Contact( "DB2120_MPP_ITC_IPC".RESET_FAULTS )
   END_RUNG wire#w1
   RUNG wire#w2
      Coil( "DB426_ALARMS_WARNINGS".ALARMS.UNIT_01.STATION_3_MEASURING."716508" )
   END_RUNG
   // the same network as SCL:
   "DB16000_OPC_UA_TRIGGER_ALARM".CLIENT.U1_STA3_MEAS.ALARMS.DATABASE_CONNECTION_A := ((("DB16001_U1_STA3_MEAS_CLIENT_INTERFACE".U01_STA3_MEAS_Read.Variable.Status = (-1)) AND "DB16001_U1_STA3_MEAS_CLIENT_INTERFACE".U01_STA3_MEAS_Read.Variable.DatabaseConnection) OR ("DB16000_OPC_UA_TRIGGER_ALARM".CLIENT.U1_STA3_MEAS.ALARMS.DATABASE_CONNECTION_A AND NOT "DB2120_MPP_ITC_IPC".RESET_FAULTS)) AND "DB7253_UNIT_1_STA_3_MEAS_ENABLE_DISABLE".ENABLED;
   "DB426_ALARMS_WARNINGS".ALARMS.UNIT_01.STATION_3_MEASURING."716508" := "DB16000_OPC_UA_TRIGGER_ALARM".CLIENT.U1_STA3_MEAS.ALARMS.DATABASE_CONNECTION_A;
END_REGION

REGION Network 49: UNIT 1 STATION 3 MEASURING MISSING CALIBRATION IN FIXTURE 1 ALARM
   RUNG wire#powerrail
      { S7_Templates := "SrcType := Int" } EQ_Contact(in1 := "DB16010_MEASURE_SENSORS_CALIBRATION_STATUS".U1_STA3_MEAS.FIXTURE_1_STATUS, in2 := 0)
      wire#w1
      I_Contact( "DB2031_CYCLES_GENERAL".CALIBRATION_CYCLE.CYCLE_SELECTED_AUX )
      I_Contact( "DB2031_CYCLES_GENERAL".CALIBRATION_CYCLE.CYCLE_SELECTED )
      Contact( "DB7253_UNIT_1_STA_3_MEAS_ENABLE_DISABLE".ENABLED )
      wire#w2
      Coil( "DB16000_OPC_UA_TRIGGER_ALARM".CLIENT.U1_STA3_MEAS.ALARMS.CALIBRATION_MISSING_FIX_1_A )
   END_RUNG
   RUNG wire#powerrail
      Contact( "DB16000_OPC_UA_TRIGGER_ALARM".CLIENT.U1_STA3_MEAS.ALARMS.CALIBRATION_MISSING_FIX_1_A )
      I_Contact( "DB2120_MPP_ITC_IPC".RESET_FAULTS )
   END_RUNG wire#w1
   RUNG wire#w2
      Coil( "DB426_ALARMS_WARNINGS".ALARMS.UNIT_01.STATION_3_MEASURING."716510" )
   END_RUNG
   // the same network as SCL:
   "DB16000_OPC_UA_TRIGGER_ALARM".CLIENT.U1_STA3_MEAS.ALARMS.CALIBRATION_MISSING_FIX_1_A := (("DB16010_MEASURE_SENSORS_CALIBRATION_STATUS".U1_STA3_MEAS.FIXTURE_1_STATUS = 0) OR ("DB16000_OPC_UA_TRIGGER_ALARM".CLIENT.U1_STA3_MEAS.ALARMS.CALIBRATION_MISSING_FIX_1_A AND NOT "DB2120_MPP_ITC_IPC".RESET_FAULTS)) AND NOT "DB2031_CYCLES_GENERAL".CALIBRATION_CYCLE.CYCLE_SELECTED_AUX AND NOT "DB2031_CYCLES_GENERAL".CALIBRATION_CYCLE.CYCLE_SELECTED AND "DB7253_UNIT_1_STA_3_MEAS_ENABLE_DISABLE".ENABLED;
   "DB426_ALARMS_WARNINGS".ALARMS.UNIT_01.STATION_3_MEASURING."716510" := "DB16000_OPC_UA_TRIGGER_ALARM".CLIENT.U1_STA3_MEAS.ALARMS.CALIBRATION_MISSING_FIX_1_A;
END_REGION

REGION Network 50: UNIT 1 STATION 3 MEASURING MISSING CALIBRATION IN FIXTURE 2 ALARM
   RUNG wire#powerrail
      { S7_Templates := "SrcType := Int" } EQ_Contact(in1 := "DB16010_MEASURE_SENSORS_CALIBRATION_STATUS".U1_STA3_MEAS.FIXTURE_2_STATUS, in2 := 0)
      wire#w1
      I_Contact( "DB2031_CYCLES_GENERAL".CALIBRATION_CYCLE.CYCLE_SELECTED_AUX )
      I_Contact( "DB2031_CYCLES_GENERAL".CALIBRATION_CYCLE.CYCLE_SELECTED )
      Contact( "DB7253_UNIT_1_STA_3_MEAS_ENABLE_DISABLE".ENABLED )
      wire#w2
      Coil( "DB16000_OPC_UA_TRIGGER_ALARM".CLIENT.U1_STA3_MEAS.ALARMS.CALIBRATION_MISSING_FIX_2_A )
   END_RUNG
   RUNG wire#powerrail
      Contact( "DB16000_OPC_UA_TRIGGER_ALARM".CLIENT.U1_STA3_MEAS.ALARMS.CALIBRATION_MISSING_FIX_2_A )
      I_Contact( "DB2120_MPP_ITC_IPC".RESET_FAULTS )
   END_RUNG wire#w1
   RUNG wire#w2
      Coil( "DB426_ALARMS_WARNINGS".ALARMS.UNIT_01.STATION_3_MEASURING."716511" )
   END_RUNG
   // the same network as SCL:
   "DB16000_OPC_UA_TRIGGER_ALARM".CLIENT.U1_STA3_MEAS.ALARMS.CALIBRATION_MISSING_FIX_2_A := (("DB16010_MEASURE_SENSORS_CALIBRATION_STATUS".U1_STA3_MEAS.FIXTURE_2_STATUS = 0) OR ("DB16000_OPC_UA_TRIGGER_ALARM".CLIENT.U1_STA3_MEAS.ALARMS.CALIBRATION_MISSING_FIX_2_A AND NOT "DB2120_MPP_ITC_IPC".RESET_FAULTS)) AND NOT "DB2031_CYCLES_GENERAL".CALIBRATION_CYCLE.CYCLE_SELECTED_AUX AND NOT "DB2031_CYCLES_GENERAL".CALIBRATION_CYCLE.CYCLE_SELECTED AND "DB7253_UNIT_1_STA_3_MEAS_ENABLE_DISABLE".ENABLED;
   "DB426_ALARMS_WARNINGS".ALARMS.UNIT_01.STATION_3_MEASURING."716511" := "DB16000_OPC_UA_TRIGGER_ALARM".CLIENT.U1_STA3_MEAS.ALARMS.CALIBRATION_MISSING_FIX_2_A;
END_REGION

REGION Network 51: UNIT 1 STATION 3 MEASURING MISSING CALIBRATION IN FIXTURE 3 ALARM
   RUNG wire#powerrail
      { S7_Templates := "SrcType := Int" } EQ_Contact(in1 := "DB16010_MEASURE_SENSORS_CALIBRATION_STATUS".U1_STA3_MEAS.FIXTURE_3_STATUS, in2 := 0)
      wire#w1
      I_Contact( "DB2031_CYCLES_GENERAL".CALIBRATION_CYCLE.CYCLE_SELECTED_AUX )
      I_Contact( "DB2031_CYCLES_GENERAL".CALIBRATION_CYCLE.CYCLE_SELECTED )
      Contact( "DB7253_UNIT_1_STA_3_MEAS_ENABLE_DISABLE".ENABLED )
      wire#w2
      Coil( "DB16000_OPC_UA_TRIGGER_ALARM".CLIENT.U1_STA3_MEAS.ALARMS.CALIBRATION_MISSING_FIX_3_A )
   END_RUNG
   RUNG wire#powerrail
      Contact( "DB16000_OPC_UA_TRIGGER_ALARM".CLIENT.U1_STA3_MEAS.ALARMS.CALIBRATION_MISSING_FIX_3_A )
      I_Contact( "DB2120_MPP_ITC_IPC".RESET_FAULTS )
   END_RUNG wire#w1
   RUNG wire#w2
      Coil( "DB426_ALARMS_WARNINGS".ALARMS.UNIT_01.STATION_3_MEASURING."716512" )
   END_RUNG
   // the same network as SCL:
   "DB16000_OPC_UA_TRIGGER_ALARM".CLIENT.U1_STA3_MEAS.ALARMS.CALIBRATION_MISSING_FIX_3_A := (("DB16010_MEASURE_SENSORS_CALIBRATION_STATUS".U1_STA3_MEAS.FIXTURE_3_STATUS = 0) OR ("DB16000_OPC_UA_TRIGGER_ALARM".CLIENT.U1_STA3_MEAS.ALARMS.CALIBRATION_MISSING_FIX_3_A AND NOT "DB2120_MPP_ITC_IPC".RESET_FAULTS)) AND NOT "DB2031_CYCLES_GENERAL".CALIBRATION_CYCLE.CYCLE_SELECTED_AUX AND NOT "DB2031_CYCLES_GENERAL".CALIBRATION_CYCLE.CYCLE_SELECTED AND "DB7253_UNIT_1_STA_3_MEAS_ENABLE_DISABLE".ENABLED;
   "DB426_ALARMS_WARNINGS".ALARMS.UNIT_01.STATION_3_MEASURING."716512" := "DB16000_OPC_UA_TRIGGER_ALARM".CLIENT.U1_STA3_MEAS.ALARMS.CALIBRATION_MISSING_FIX_3_A;
END_REGION

REGION Network 52: UNIT 1 STATION 3 MEASURING MISSING CALIBRATION IN FIXTURE 4 ALARM
   RUNG wire#powerrail
      { S7_Templates := "SrcType := Int" } EQ_Contact(in1 := "DB16010_MEASURE_SENSORS_CALIBRATION_STATUS".U1_STA3_MEAS.FIXTURE_4_STATUS, in2 := 0)
      wire#w1
      I_Contact( "DB2031_CYCLES_GENERAL".CALIBRATION_CYCLE.CYCLE_SELECTED_AUX )
      I_Contact( "DB2031_CYCLES_GENERAL".CALIBRATION_CYCLE.CYCLE_SELECTED )
      Contact( "DB7253_UNIT_1_STA_3_MEAS_ENABLE_DISABLE".ENABLED )
      wire#w2
      Coil( "DB16000_OPC_UA_TRIGGER_ALARM".CLIENT.U1_STA3_MEAS.ALARMS.CALIBRATION_MISSING_FIX_4_A )
   END_RUNG
   RUNG wire#powerrail
      Contact( "DB16000_OPC_UA_TRIGGER_ALARM".CLIENT.U1_STA3_MEAS.ALARMS.CALIBRATION_MISSING_FIX_4_A )
      I_Contact( "DB2120_MPP_ITC_IPC".RESET_FAULTS )
   END_RUNG wire#w1
   RUNG wire#w2
      Coil( "DB426_ALARMS_WARNINGS".ALARMS.UNIT_01.STATION_3_MEASURING."716513" )
   END_RUNG
   // the same network as SCL:
   "DB16000_OPC_UA_TRIGGER_ALARM".CLIENT.U1_STA3_MEAS.ALARMS.CALIBRATION_MISSING_FIX_4_A := (("DB16010_MEASURE_SENSORS_CALIBRATION_STATUS".U1_STA3_MEAS.FIXTURE_4_STATUS = 0) OR ("DB16000_OPC_UA_TRIGGER_ALARM".CLIENT.U1_STA3_MEAS.ALARMS.CALIBRATION_MISSING_FIX_4_A AND NOT "DB2120_MPP_ITC_IPC".RESET_FAULTS)) AND NOT "DB2031_CYCLES_GENERAL".CALIBRATION_CYCLE.CYCLE_SELECTED_AUX AND NOT "DB2031_CYCLES_GENERAL".CALIBRATION_CYCLE.CYCLE_SELECTED AND "DB7253_UNIT_1_STA_3_MEAS_ENABLE_DISABLE".ENABLED;
   "DB426_ALARMS_WARNINGS".ALARMS.UNIT_01.STATION_3_MEASURING."716513" := "DB16000_OPC_UA_TRIGGER_ALARM".CLIENT.U1_STA3_MEAS.ALARMS.CALIBRATION_MISSING_FIX_4_A;
END_REGION

REGION Network 53: UNIT 1 STATION 3 MEASURING LAST CALIBRATION OUT OF RANGE IN FIXTURE 1 ALARM----------
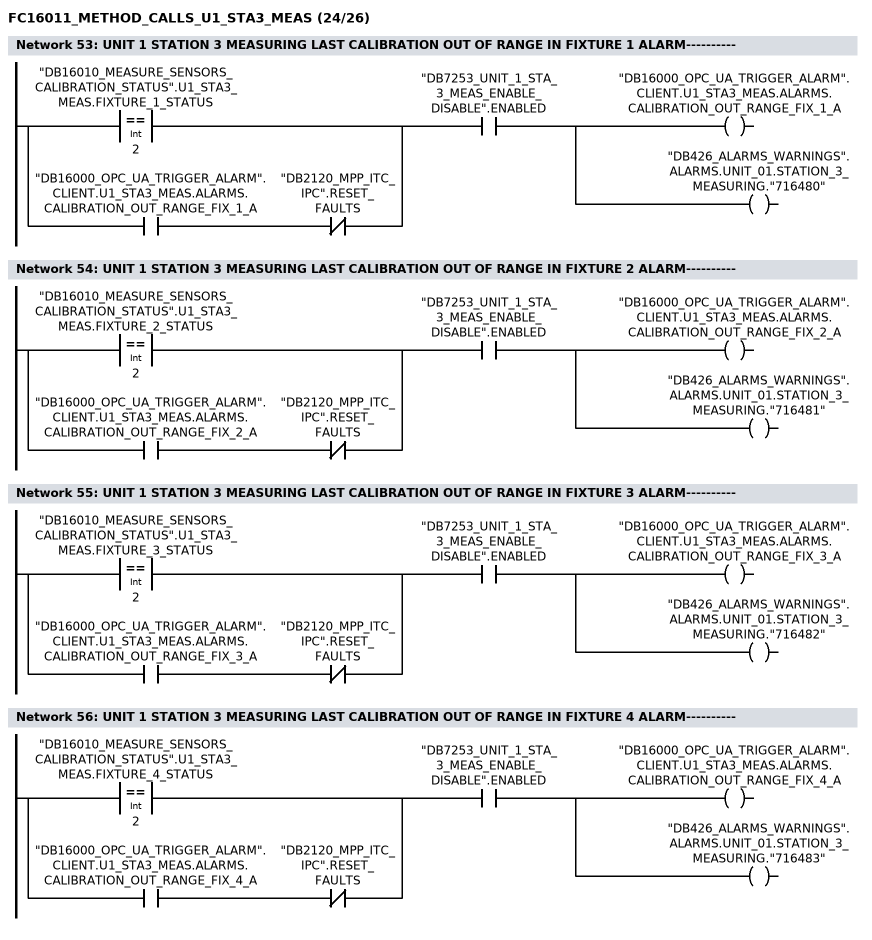
   RUNG wire#powerrail
      { S7_Templates := "SrcType := Int" } EQ_Contact(in1 := "DB16010_MEASURE_SENSORS_CALIBRATION_STATUS".U1_STA3_MEAS.FIXTURE_1_STATUS, in2 := 2)
      wire#w1
      Contact( "DB7253_UNIT_1_STA_3_MEAS_ENABLE_DISABLE".ENABLED )
      wire#w2
      Coil( "DB16000_OPC_UA_TRIGGER_ALARM".CLIENT.U1_STA3_MEAS.ALARMS.CALIBRATION_OUT_RANGE_FIX_1_A )
   END_RUNG
   RUNG wire#powerrail
      Contact( "DB16000_OPC_UA_TRIGGER_ALARM".CLIENT.U1_STA3_MEAS.ALARMS.CALIBRATION_OUT_RANGE_FIX_1_A )
      I_Contact( "DB2120_MPP_ITC_IPC".RESET_FAULTS )
   END_RUNG wire#w1
   RUNG wire#w2
      Coil( "DB426_ALARMS_WARNINGS".ALARMS.UNIT_01.STATION_3_MEASURING."716480" )
   END_RUNG
   // the same network as SCL:
   "DB16000_OPC_UA_TRIGGER_ALARM".CLIENT.U1_STA3_MEAS.ALARMS.CALIBRATION_OUT_RANGE_FIX_1_A := (("DB16010_MEASURE_SENSORS_CALIBRATION_STATUS".U1_STA3_MEAS.FIXTURE_1_STATUS = 2) OR ("DB16000_OPC_UA_TRIGGER_ALARM".CLIENT.U1_STA3_MEAS.ALARMS.CALIBRATION_OUT_RANGE_FIX_1_A AND NOT "DB2120_MPP_ITC_IPC".RESET_FAULTS)) AND "DB7253_UNIT_1_STA_3_MEAS_ENABLE_DISABLE".ENABLED;
   "DB426_ALARMS_WARNINGS".ALARMS.UNIT_01.STATION_3_MEASURING."716480" := "DB16000_OPC_UA_TRIGGER_ALARM".CLIENT.U1_STA3_MEAS.ALARMS.CALIBRATION_OUT_RANGE_FIX_1_A;
END_REGION

REGION Network 54: UNIT 1 STATION 3 MEASURING LAST CALIBRATION OUT OF RANGE IN FIXTURE 2 ALARM----------
   RUNG wire#powerrail
      { S7_Templates := "SrcType := Int" } EQ_Contact(in1 := "DB16010_MEASURE_SENSORS_CALIBRATION_STATUS".U1_STA3_MEAS.FIXTURE_2_STATUS, in2 := 2)
      wire#w1
      Contact( "DB7253_UNIT_1_STA_3_MEAS_ENABLE_DISABLE".ENABLED )
      wire#w2
      Coil( "DB16000_OPC_UA_TRIGGER_ALARM".CLIENT.U1_STA3_MEAS.ALARMS.CALIBRATION_OUT_RANGE_FIX_2_A )
   END_RUNG
   RUNG wire#powerrail
      Contact( "DB16000_OPC_UA_TRIGGER_ALARM".CLIENT.U1_STA3_MEAS.ALARMS.CALIBRATION_OUT_RANGE_FIX_2_A )
      I_Contact( "DB2120_MPP_ITC_IPC".RESET_FAULTS )
   END_RUNG wire#w1
   RUNG wire#w2
      Coil( "DB426_ALARMS_WARNINGS".ALARMS.UNIT_01.STATION_3_MEASURING."716481" )
   END_RUNG
   // the same network as SCL:
   "DB16000_OPC_UA_TRIGGER_ALARM".CLIENT.U1_STA3_MEAS.ALARMS.CALIBRATION_OUT_RANGE_FIX_2_A := (("DB16010_MEASURE_SENSORS_CALIBRATION_STATUS".U1_STA3_MEAS.FIXTURE_2_STATUS = 2) OR ("DB16000_OPC_UA_TRIGGER_ALARM".CLIENT.U1_STA3_MEAS.ALARMS.CALIBRATION_OUT_RANGE_FIX_2_A AND NOT "DB2120_MPP_ITC_IPC".RESET_FAULTS)) AND "DB7253_UNIT_1_STA_3_MEAS_ENABLE_DISABLE".ENABLED;
   "DB426_ALARMS_WARNINGS".ALARMS.UNIT_01.STATION_3_MEASURING."716481" := "DB16000_OPC_UA_TRIGGER_ALARM".CLIENT.U1_STA3_MEAS.ALARMS.CALIBRATION_OUT_RANGE_FIX_2_A;
END_REGION

REGION Network 55: UNIT 1 STATION 3 MEASURING LAST CALIBRATION OUT OF RANGE IN FIXTURE 3 ALARM----------
   RUNG wire#powerrail
      { S7_Templates := "SrcType := Int" } EQ_Contact(in1 := "DB16010_MEASURE_SENSORS_CALIBRATION_STATUS".U1_STA3_MEAS.FIXTURE_3_STATUS, in2 := 2)
      wire#w1
      Contact( "DB7253_UNIT_1_STA_3_MEAS_ENABLE_DISABLE".ENABLED )
      wire#w2
      Coil( "DB16000_OPC_UA_TRIGGER_ALARM".CLIENT.U1_STA3_MEAS.ALARMS.CALIBRATION_OUT_RANGE_FIX_3_A )
   END_RUNG
   RUNG wire#powerrail
      Contact( "DB16000_OPC_UA_TRIGGER_ALARM".CLIENT.U1_STA3_MEAS.ALARMS.CALIBRATION_OUT_RANGE_FIX_3_A )
      I_Contact( "DB2120_MPP_ITC_IPC".RESET_FAULTS )
   END_RUNG wire#w1
   RUNG wire#w2
      Coil( "DB426_ALARMS_WARNINGS".ALARMS.UNIT_01.STATION_3_MEASURING."716482" )
   END_RUNG
   // the same network as SCL:
   "DB16000_OPC_UA_TRIGGER_ALARM".CLIENT.U1_STA3_MEAS.ALARMS.CALIBRATION_OUT_RANGE_FIX_3_A := (("DB16010_MEASURE_SENSORS_CALIBRATION_STATUS".U1_STA3_MEAS.FIXTURE_3_STATUS = 2) OR ("DB16000_OPC_UA_TRIGGER_ALARM".CLIENT.U1_STA3_MEAS.ALARMS.CALIBRATION_OUT_RANGE_FIX_3_A AND NOT "DB2120_MPP_ITC_IPC".RESET_FAULTS)) AND "DB7253_UNIT_1_STA_3_MEAS_ENABLE_DISABLE".ENABLED;
   "DB426_ALARMS_WARNINGS".ALARMS.UNIT_01.STATION_3_MEASURING."716482" := "DB16000_OPC_UA_TRIGGER_ALARM".CLIENT.U1_STA3_MEAS.ALARMS.CALIBRATION_OUT_RANGE_FIX_3_A;
END_REGION

REGION Network 56: UNIT 1 STATION 3 MEASURING LAST CALIBRATION OUT OF RANGE IN FIXTURE 4 ALARM----------
   RUNG wire#powerrail
      { S7_Templates := "SrcType := Int" } EQ_Contact(in1 := "DB16010_MEASURE_SENSORS_CALIBRATION_STATUS".U1_STA3_MEAS.FIXTURE_4_STATUS, in2 := 2)
      wire#w1
      Contact( "DB7253_UNIT_1_STA_3_MEAS_ENABLE_DISABLE".ENABLED )
      wire#w2
      Coil( "DB16000_OPC_UA_TRIGGER_ALARM".CLIENT.U1_STA3_MEAS.ALARMS.CALIBRATION_OUT_RANGE_FIX_4_A )
   END_RUNG
   RUNG wire#powerrail
      Contact( "DB16000_OPC_UA_TRIGGER_ALARM".CLIENT.U1_STA3_MEAS.ALARMS.CALIBRATION_OUT_RANGE_FIX_4_A )
      I_Contact( "DB2120_MPP_ITC_IPC".RESET_FAULTS )
   END_RUNG wire#w1
   RUNG wire#w2
      Coil( "DB426_ALARMS_WARNINGS".ALARMS.UNIT_01.STATION_3_MEASURING."716483" )
   END_RUNG
   // the same network as SCL:
   "DB16000_OPC_UA_TRIGGER_ALARM".CLIENT.U1_STA3_MEAS.ALARMS.CALIBRATION_OUT_RANGE_FIX_4_A := (("DB16010_MEASURE_SENSORS_CALIBRATION_STATUS".U1_STA3_MEAS.FIXTURE_4_STATUS = 2) OR ("DB16000_OPC_UA_TRIGGER_ALARM".CLIENT.U1_STA3_MEAS.ALARMS.CALIBRATION_OUT_RANGE_FIX_4_A AND NOT "DB2120_MPP_ITC_IPC".RESET_FAULTS)) AND "DB7253_UNIT_1_STA_3_MEAS_ENABLE_DISABLE".ENABLED;
   "DB426_ALARMS_WARNINGS".ALARMS.UNIT_01.STATION_3_MEASURING."716483" := "DB16000_OPC_UA_TRIGGER_ALARM".CLIENT.U1_STA3_MEAS.ALARMS.CALIBRATION_OUT_RANGE_FIX_4_A;
END_REGION

REGION Network 57: UNIT 1 STATION 3 MEASURING CALIBRATION PROCEDURE ALARM
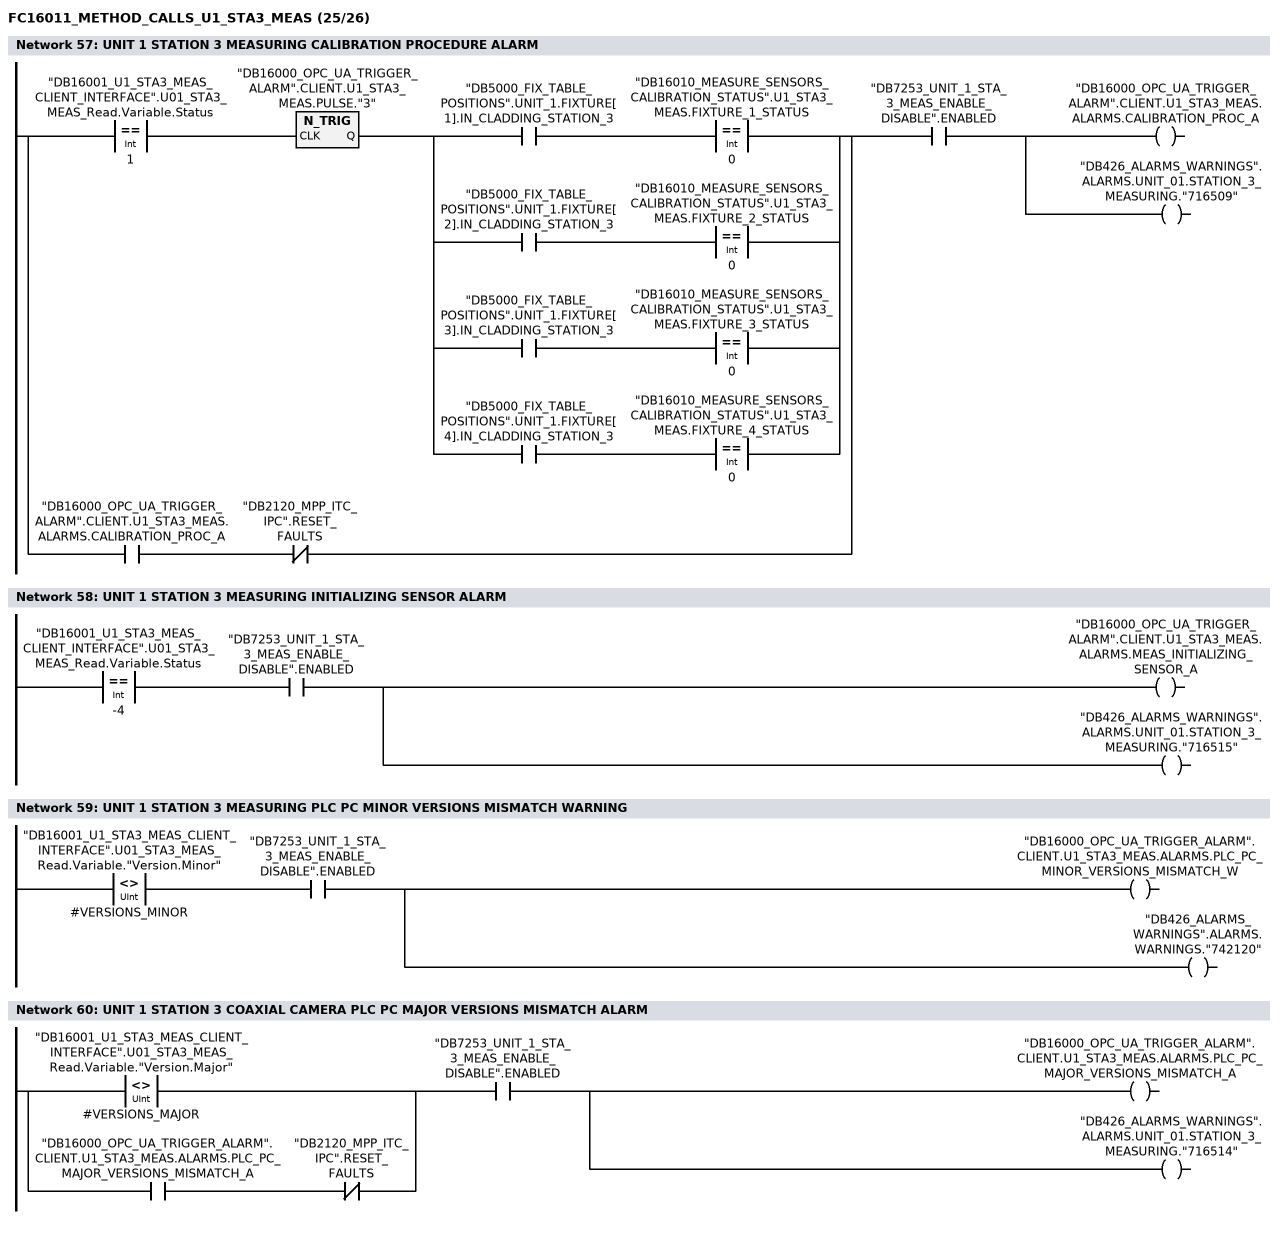
   RUNG wire#powerrail
      { S7_Templates := "SrcType := Int" } EQ_Contact(in1 := "DB16001_U1_STA3_MEAS_CLIENT_INTERFACE".U01_STA3_MEAS_Read.Variable.Status, in2 := 1)
      N_Trig( "DB16000_OPC_UA_TRIGGER_ALARM".CLIENT.U1_STA3_MEAS.PULSE."3" )
      wire#w1
      Contact( "DB5000_FIX_TABLE_POSITIONS".UNIT_1.FIXTURE[1].IN_CLADDING_STATION_3 )
      { S7_Templates := "SrcType := Int" } EQ_Contact(in1 := "DB16010_MEASURE_SENSORS_CALIBRATION_STATUS".U1_STA3_MEAS.FIXTURE_1_STATUS, in2 := 0)
      wire#w2
      Contact( "DB7253_UNIT_1_STA_3_MEAS_ENABLE_DISABLE".ENABLED )
      wire#w3
      Coil( "DB16000_OPC_UA_TRIGGER_ALARM".CLIENT.U1_STA3_MEAS.ALARMS.CALIBRATION_PROC_A )
   END_RUNG
   RUNG wire#w1
      Contact( "DB5000_FIX_TABLE_POSITIONS".UNIT_1.FIXTURE[2].IN_CLADDING_STATION_3 )
      { S7_Templates := "SrcType := Int" } EQ_Contact(in1 := "DB16010_MEASURE_SENSORS_CALIBRATION_STATUS".U1_STA3_MEAS.FIXTURE_2_STATUS, in2 := 0)
   END_RUNG wire#w2
   RUNG wire#w1
      Contact( "DB5000_FIX_TABLE_POSITIONS".UNIT_1.FIXTURE[3].IN_CLADDING_STATION_3 )
      { S7_Templates := "SrcType := Int" } EQ_Contact(in1 := "DB16010_MEASURE_SENSORS_CALIBRATION_STATUS".U1_STA3_MEAS.FIXTURE_3_STATUS, in2 := 0)
   END_RUNG wire#w2
   RUNG wire#w1
      Contact( "DB5000_FIX_TABLE_POSITIONS".UNIT_1.FIXTURE[4].IN_CLADDING_STATION_3 )
      { S7_Templates := "SrcType := Int" } EQ_Contact(in1 := "DB16010_MEASURE_SENSORS_CALIBRATION_STATUS".U1_STA3_MEAS.FIXTURE_4_STATUS, in2 := 0)
   END_RUNG wire#w2
   RUNG wire#powerrail
      Contact( "DB16000_OPC_UA_TRIGGER_ALARM".CLIENT.U1_STA3_MEAS.ALARMS.CALIBRATION_PROC_A )
      I_Contact( "DB2120_MPP_ITC_IPC".RESET_FAULTS )
   END_RUNG wire#w2
   RUNG wire#w3
      Coil( "DB426_ALARMS_WARNINGS".ALARMS.UNIT_01.STATION_3_MEASURING."716509" )
   END_RUNG
   // the same network as SCL:
   #_w1 := "DB16001_U1_STA3_MEAS_CLIENT_INTERFACE".U01_STA3_MEAS_Read.Variable.Status = 1;
   #_w2 := NOT #_w1 AND "DB16000_OPC_UA_TRIGGER_ALARM".CLIENT.U1_STA3_MEAS.PULSE."3";   // falling edge
   "DB16000_OPC_UA_TRIGGER_ALARM".CLIENT.U1_STA3_MEAS.PULSE."3" := #_w1;
   "DB16000_OPC_UA_TRIGGER_ALARM".CLIENT.U1_STA3_MEAS.ALARMS.CALIBRATION_PROC_A := ((#_w2 AND (("DB5000_FIX_TABLE_POSITIONS".UNIT_1.FIXTURE[1].IN_CLADDING_STATION_3 AND ("DB16010_MEASURE_SENSORS_CALIBRATION_STATUS".U1_STA3_MEAS.FIXTURE_1_STATUS = 0)) OR ("DB5000_FIX_TABLE_POSITIONS".UNIT_1.FIXTURE[2].IN_CLADDING_STATION_3 AND ("DB16010_MEASURE_SENSORS_CALIBRATION_STATUS".U1_STA3_MEAS.FIXTURE_2_STATUS = 0)) OR ("DB5000_FIX_TABLE_POSITIONS".UNIT_1.FIXTURE[3].IN_CLADDING_STATION_3 AND ("DB16010_MEASURE_SENSORS_CALIBRATION_STATUS".U1_STA3_MEAS.FIXTURE_3_STATUS = 0)) OR ("DB5000_FIX_TABLE_POSITIONS".UNIT_1.FIXTURE[4].IN_CLADDING_STATION_3 AND ("DB16010_MEASURE_SENSORS_CALIBRATION_STATUS".U1_STA3_MEAS.FIXTURE_4_STATUS = 0)))) OR ("DB16000_OPC_UA_TRIGGER_ALARM".CLIENT.U1_STA3_MEAS.ALARMS.CALIBRATION_PROC_A AND NOT "DB2120_MPP_ITC_IPC".RESET_FAULTS)) AND "DB7253_UNIT_1_STA_3_MEAS_ENABLE_DISABLE".ENABLED;
   "DB426_ALARMS_WARNINGS".ALARMS.UNIT_01.STATION_3_MEASURING."716509" := "DB16000_OPC_UA_TRIGGER_ALARM".CLIENT.U1_STA3_MEAS.ALARMS.CALIBRATION_PROC_A;
END_REGION

REGION Network 58: UNIT 1 STATION 3 MEASURING INITIALIZING SENSOR ALARM
   RUNG wire#powerrail
      { S7_Templates := "SrcType := Int" } EQ_Contact(in1 := "DB16001_U1_STA3_MEAS_CLIENT_INTERFACE".U01_STA3_MEAS_Read.Variable.Status, in2 := -4)
      Contact( "DB7253_UNIT_1_STA_3_MEAS_ENABLE_DISABLE".ENABLED )
      wire#w1
      Coil( "DB16000_OPC_UA_TRIGGER_ALARM".CLIENT.U1_STA3_MEAS.ALARMS.MEAS_INITIALIZING_SENSOR_A )
   END_RUNG
   RUNG wire#w1
      Coil( "DB426_ALARMS_WARNINGS".ALARMS.UNIT_01.STATION_3_MEASURING."716515" )
   END_RUNG
   // the same network as SCL:
   "DB16000_OPC_UA_TRIGGER_ALARM".CLIENT.U1_STA3_MEAS.ALARMS.MEAS_INITIALIZING_SENSOR_A := ("DB16001_U1_STA3_MEAS_CLIENT_INTERFACE".U01_STA3_MEAS_Read.Variable.Status = (-4)) AND "DB7253_UNIT_1_STA_3_MEAS_ENABLE_DISABLE".ENABLED;
   "DB426_ALARMS_WARNINGS".ALARMS.UNIT_01.STATION_3_MEASURING."716515" := "DB16000_OPC_UA_TRIGGER_ALARM".CLIENT.U1_STA3_MEAS.ALARMS.MEAS_INITIALIZING_SENSOR_A;
END_REGION

REGION Network 59: UNIT 1 STATION 3 MEASURING PLC PC MINOR VERSIONS MISMATCH WARNING
   RUNG wire#powerrail
      { S7_Templates := "SrcType := UInt" } NE_Contact(in1 := "DB16001_U1_STA3_MEAS_CLIENT_INTERFACE".U01_STA3_MEAS_Read.Variable."Version.Minor", in2 := #VERSIONS_MINOR)
      Contact( "DB7253_UNIT_1_STA_3_MEAS_ENABLE_DISABLE".ENABLED )
      wire#w1
      Coil( "DB16000_OPC_UA_TRIGGER_ALARM".CLIENT.U1_STA3_MEAS.ALARMS.PLC_PC_MINOR_VERSIONS_MISMATCH_W )
   END_RUNG
   RUNG wire#w1
      Coil( "DB426_ALARMS_WARNINGS".ALARMS.WARNINGS."742120" )
   END_RUNG
   // the same network as SCL:
   "DB16000_OPC_UA_TRIGGER_ALARM".CLIENT.U1_STA3_MEAS.ALARMS.PLC_PC_MINOR_VERSIONS_MISMATCH_W := ("DB16001_U1_STA3_MEAS_CLIENT_INTERFACE".U01_STA3_MEAS_Read.Variable."Version.Minor" <> #VERSIONS_MINOR) AND "DB7253_UNIT_1_STA_3_MEAS_ENABLE_DISABLE".ENABLED;
   "DB426_ALARMS_WARNINGS".ALARMS.WARNINGS."742120" := "DB16000_OPC_UA_TRIGGER_ALARM".CLIENT.U1_STA3_MEAS.ALARMS.PLC_PC_MINOR_VERSIONS_MISMATCH_W;
END_REGION

REGION Network 60: UNIT 1 STATION 3 COAXIAL CAMERA PLC PC MAJOR VERSIONS MISMATCH ALARM
   RUNG wire#powerrail
      { S7_Templates := "SrcType := UInt" } NE_Contact(in1 := "DB16001_U1_STA3_MEAS_CLIENT_INTERFACE".U01_STA3_MEAS_Read.Variable."Version.Major", in2 := #VERSIONS_MAJOR)
      wire#w1
      Contact( "DB7253_UNIT_1_STA_3_MEAS_ENABLE_DISABLE".ENABLED )
      wire#w2
      Coil( "DB16000_OPC_UA_TRIGGER_ALARM".CLIENT.U1_STA3_MEAS.ALARMS.PLC_PC_MAJOR_VERSIONS_MISMATCH_A )
   END_RUNG
   RUNG wire#powerrail
      Contact( "DB16000_OPC_UA_TRIGGER_ALARM".CLIENT.U1_STA3_MEAS.ALARMS.PLC_PC_MAJOR_VERSIONS_MISMATCH_A )
      I_Contact( "DB2120_MPP_ITC_IPC".RESET_FAULTS )
   END_RUNG wire#w1
   RUNG wire#w2
      Coil( "DB426_ALARMS_WARNINGS".ALARMS.UNIT_01.STATION_3_MEASURING."716514" )
   END_RUNG
   // the same network as SCL:
   "DB16000_OPC_UA_TRIGGER_ALARM".CLIENT.U1_STA3_MEAS.ALARMS.PLC_PC_MAJOR_VERSIONS_MISMATCH_A := (("DB16001_U1_STA3_MEAS_CLIENT_INTERFACE".U01_STA3_MEAS_Read.Variable."Version.Major" <> #VERSIONS_MAJOR) OR ("DB16000_OPC_UA_TRIGGER_ALARM".CLIENT.U1_STA3_MEAS.ALARMS.PLC_PC_MAJOR_VERSIONS_MISMATCH_A AND NOT "DB2120_MPP_ITC_IPC".RESET_FAULTS)) AND "DB7253_UNIT_1_STA_3_MEAS_ENABLE_DISABLE".ENABLED;
   "DB426_ALARMS_WARNINGS".ALARMS.UNIT_01.STATION_3_MEASURING."716514" := "DB16000_OPC_UA_TRIGGER_ALARM".CLIENT.U1_STA3_MEAS.ALARMS.PLC_PC_MAJOR_VERSIONS_MISMATCH_A;
END_REGION

REGION Network 61: IS_SEOC ALARMS
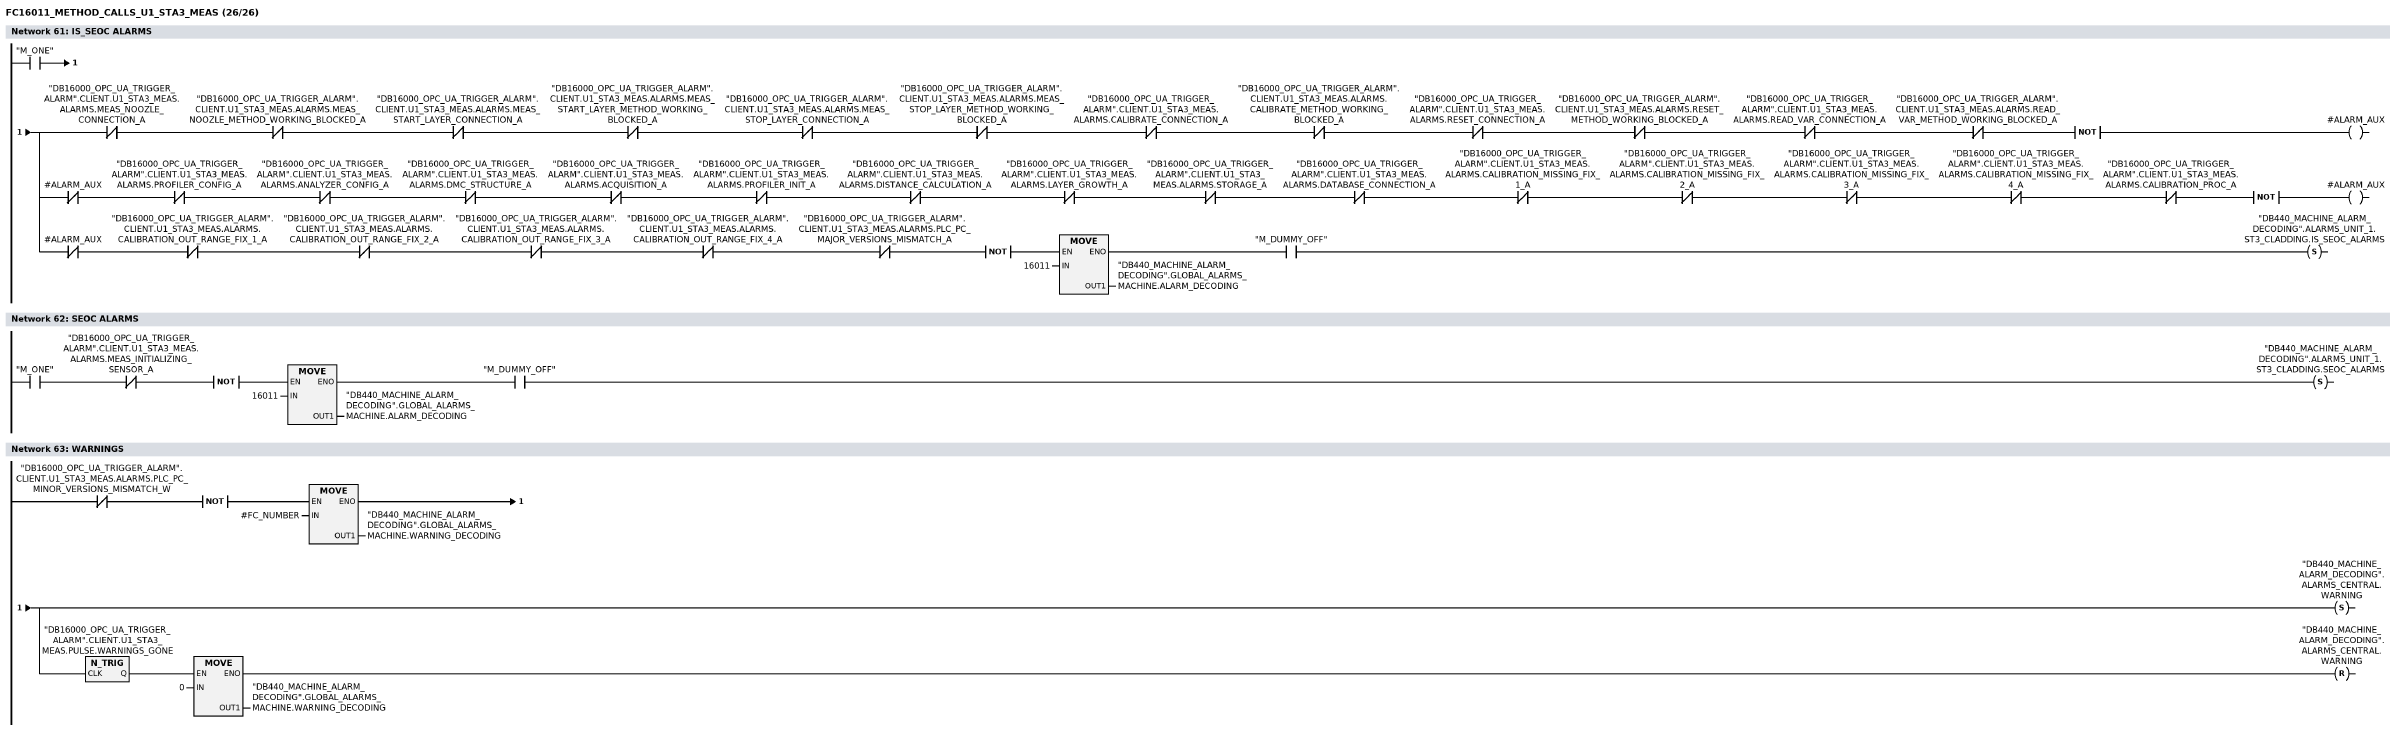
   RUNG wire#powerrail
      Contact( "M_ONE" )
      wire#w1
      I_Contact( "DB16000_OPC_UA_TRIGGER_ALARM".CLIENT.U1_STA3_MEAS.ALARMS.MEAS_NOOZLE_CONNECTION_A )
      I_Contact( "DB16000_OPC_UA_TRIGGER_ALARM".CLIENT.U1_STA3_MEAS.ALARMS.MEAS_NOOZLE_METHOD_WORKING_BLOCKED_A )
      I_Contact( "DB16000_OPC_UA_TRIGGER_ALARM".CLIENT.U1_STA3_MEAS.ALARMS.MEAS_START_LAYER_CONNECTION_A )
      I_Contact( "DB16000_OPC_UA_TRIGGER_ALARM".CLIENT.U1_STA3_MEAS.ALARMS.MEAS_START_LAYER_METHOD_WORKING_BLOCKED_A )
      I_Contact( "DB16000_OPC_UA_TRIGGER_ALARM".CLIENT.U1_STA3_MEAS.ALARMS.MEAS_STOP_LAYER_CONNECTION_A )
      I_Contact( "DB16000_OPC_UA_TRIGGER_ALARM".CLIENT.U1_STA3_MEAS.ALARMS.MEAS_STOP_LAYER_METHOD_WORKING_BLOCKED_A )
      I_Contact( "DB16000_OPC_UA_TRIGGER_ALARM".CLIENT.U1_STA3_MEAS.ALARMS.CALIBRATE_CONNECTION_A )
      I_Contact( "DB16000_OPC_UA_TRIGGER_ALARM".CLIENT.U1_STA3_MEAS.ALARMS.CALIBRATE_METHOD_WORKING_BLOCKED_A )
      I_Contact( "DB16000_OPC_UA_TRIGGER_ALARM".CLIENT.U1_STA3_MEAS.ALARMS.RESET_CONNECTION_A )
      I_Contact( "DB16000_OPC_UA_TRIGGER_ALARM".CLIENT.U1_STA3_MEAS.ALARMS.RESET_METHOD_WORKING_BLOCKED_A )
      I_Contact( "DB16000_OPC_UA_TRIGGER_ALARM".CLIENT.U1_STA3_MEAS.ALARMS.READ_VAR_CONNECTION_A )
      I_Contact( "DB16000_OPC_UA_TRIGGER_ALARM".CLIENT.U1_STA3_MEAS.ALARMS.READ_VAR_METHOD_WORKING_BLOCKED_A )
      Not()
      Coil( #ALARM_AUX )
   END_RUNG
   RUNG wire#w1
      I_Contact( #ALARM_AUX )
      I_Contact( "DB16000_OPC_UA_TRIGGER_ALARM".CLIENT.U1_STA3_MEAS.ALARMS.PROFILER_CONFIG_A )
      I_Contact( "DB16000_OPC_UA_TRIGGER_ALARM".CLIENT.U1_STA3_MEAS.ALARMS.ANALYZER_CONFIG_A )
      I_Contact( "DB16000_OPC_UA_TRIGGER_ALARM".CLIENT.U1_STA3_MEAS.ALARMS.DMC_STRUCTURE_A )
      I_Contact( "DB16000_OPC_UA_TRIGGER_ALARM".CLIENT.U1_STA3_MEAS.ALARMS.ACQUISITION_A )
      I_Contact( "DB16000_OPC_UA_TRIGGER_ALARM".CLIENT.U1_STA3_MEAS.ALARMS.PROFILER_INIT_A )
      I_Contact( "DB16000_OPC_UA_TRIGGER_ALARM".CLIENT.U1_STA3_MEAS.ALARMS.DISTANCE_CALCULATION_A )
      I_Contact( "DB16000_OPC_UA_TRIGGER_ALARM".CLIENT.U1_STA3_MEAS.ALARMS.LAYER_GROWTH_A )
      I_Contact( "DB16000_OPC_UA_TRIGGER_ALARM".CLIENT.U1_STA3_MEAS.ALARMS.STORAGE_A )
      I_Contact( "DB16000_OPC_UA_TRIGGER_ALARM".CLIENT.U1_STA3_MEAS.ALARMS.DATABASE_CONNECTION_A )
      I_Contact( "DB16000_OPC_UA_TRIGGER_ALARM".CLIENT.U1_STA3_MEAS.ALARMS.CALIBRATION_MISSING_FIX_1_A )
      I_Contact( "DB16000_OPC_UA_TRIGGER_ALARM".CLIENT.U1_STA3_MEAS.ALARMS.CALIBRATION_MISSING_FIX_2_A )
      I_Contact( "DB16000_OPC_UA_TRIGGER_ALARM".CLIENT.U1_STA3_MEAS.ALARMS.CALIBRATION_MISSING_FIX_3_A )
      I_Contact( "DB16000_OPC_UA_TRIGGER_ALARM".CLIENT.U1_STA3_MEAS.ALARMS.CALIBRATION_MISSING_FIX_4_A )
      I_Contact( "DB16000_OPC_UA_TRIGGER_ALARM".CLIENT.U1_STA3_MEAS.ALARMS.CALIBRATION_PROC_A )
      Not()
      Coil( #ALARM_AUX )
   END_RUNG
   RUNG wire#w1
      I_Contact( #ALARM_AUX )
      I_Contact( "DB16000_OPC_UA_TRIGGER_ALARM".CLIENT.U1_STA3_MEAS.ALARMS.CALIBRATION_OUT_RANGE_FIX_1_A )
      I_Contact( "DB16000_OPC_UA_TRIGGER_ALARM".CLIENT.U1_STA3_MEAS.ALARMS.CALIBRATION_OUT_RANGE_FIX_2_A )
      I_Contact( "DB16000_OPC_UA_TRIGGER_ALARM".CLIENT.U1_STA3_MEAS.ALARMS.CALIBRATION_OUT_RANGE_FIX_3_A )
      I_Contact( "DB16000_OPC_UA_TRIGGER_ALARM".CLIENT.U1_STA3_MEAS.ALARMS.CALIBRATION_OUT_RANGE_FIX_4_A )
      I_Contact( "DB16000_OPC_UA_TRIGGER_ALARM".CLIENT.U1_STA3_MEAS.ALARMS.PLC_PC_MAJOR_VERSIONS_MISMATCH_A )
      Not()
      Move(in := 16011, out1 => "DB440_MACHINE_ALARM_DECODING".GLOBAL_ALARMS_MACHINE.ALARM_DECODING)
      Contact( "M_DUMMY_OFF" )
      S_Coil( "DB440_MACHINE_ALARM_DECODING".ALARMS_UNIT_1.ST3_CLADDING.IS_SEOC_ALARMS )
   END_RUNG
   // the same network as SCL:
   #ALARM_AUX := NOT ("M_ONE" AND NOT "DB16000_OPC_UA_TRIGGER_ALARM".CLIENT.U1_STA3_MEAS.ALARMS.MEAS_NOOZLE_CONNECTION_A AND NOT "DB16000_OPC_UA_TRIGGER_ALARM".CLIENT.U1_STA3_MEAS.ALARMS.MEAS_NOOZLE_METHOD_WORKING_BLOCKED_A AND NOT "DB16000_OPC_UA_TRIGGER_ALARM".CLIENT.U1_STA3_MEAS.ALARMS.MEAS_START_LAYER_CONNECTION_A AND NOT "DB16000_OPC_UA_TRIGGER_ALARM".CLIENT.U1_STA3_MEAS.ALARMS.MEAS_START_LAYER_METHOD_WORKING_BLOCKED_A AND NOT "DB16000_OPC_UA_TRIGGER_ALARM".CLIENT.U1_STA3_MEAS.ALARMS.MEAS_STOP_LAYER_CONNECTION_A AND NOT "DB16000_OPC_UA_TRIGGER_ALARM".CLIENT.U1_STA3_MEAS.ALARMS.MEAS_STOP_LAYER_METHOD_WORKING_BLOCKED_A AND NOT "DB16000_OPC_UA_TRIGGER_ALARM".CLIENT.U1_STA3_MEAS.ALARMS.CALIBRATE_CONNECTION_A AND NOT "DB16000_OPC_UA_TRIGGER_ALARM".CLIENT.U1_STA3_MEAS.ALARMS.CALIBRATE_METHOD_WORKING_BLOCKED_A AND NOT "DB16000_OPC_UA_TRIGGER_ALARM".CLIENT.U1_STA3_MEAS.ALARMS.RESET_CONNECTION_A AND NOT "DB16000_OPC_UA_TRIGGER_ALARM".CLIENT.U1_STA3_MEAS.ALARMS.RESET_METHOD_WORKING_BLOCKED_A AND NOT "DB16000_OPC_UA_TRIGGER_ALARM".CLIENT.U1_STA3_MEAS.ALARMS.READ_VAR_CONNECTION_A AND NOT "DB16000_OPC_UA_TRIGGER_ALARM".CLIENT.U1_STA3_MEAS.ALARMS.READ_VAR_METHOD_WORKING_BLOCKED_A);
   #ALARM_AUX := NOT ("M_ONE" AND NOT #ALARM_AUX AND NOT "DB16000_OPC_UA_TRIGGER_ALARM".CLIENT.U1_STA3_MEAS.ALARMS.PROFILER_CONFIG_A AND NOT "DB16000_OPC_UA_TRIGGER_ALARM".CLIENT.U1_STA3_MEAS.ALARMS.ANALYZER_CONFIG_A AND NOT "DB16000_OPC_UA_TRIGGER_ALARM".CLIENT.U1_STA3_MEAS.ALARMS.DMC_STRUCTURE_A AND NOT "DB16000_OPC_UA_TRIGGER_ALARM".CLIENT.U1_STA3_MEAS.ALARMS.ACQUISITION_A AND NOT "DB16000_OPC_UA_TRIGGER_ALARM".CLIENT.U1_STA3_MEAS.ALARMS.PROFILER_INIT_A AND NOT "DB16000_OPC_UA_TRIGGER_ALARM".CLIENT.U1_STA3_MEAS.ALARMS.DISTANCE_CALCULATION_A AND NOT "DB16000_OPC_UA_TRIGGER_ALARM".CLIENT.U1_STA3_MEAS.ALARMS.LAYER_GROWTH_A AND NOT "DB16000_OPC_UA_TRIGGER_ALARM".CLIENT.U1_STA3_MEAS.ALARMS.STORAGE_A AND NOT "DB16000_OPC_UA_TRIGGER_ALARM".CLIENT.U1_STA3_MEAS.ALARMS.DATABASE_CONNECTION_A AND NOT "DB16000_OPC_UA_TRIGGER_ALARM".CLIENT.U1_STA3_MEAS.ALARMS.CALIBRATION_MISSING_FIX_1_A AND NOT "DB16000_OPC_UA_TRIGGER_ALARM".CLIENT.U1_STA3_MEAS.ALARMS.CALIBRATION_MISSING_FIX_2_A AND NOT "DB16000_OPC_UA_TRIGGER_ALARM".CLIENT.U1_STA3_MEAS.ALARMS.CALIBRATION_MISSING_FIX_3_A AND NOT "DB16000_OPC_UA_TRIGGER_ALARM".CLIENT.U1_STA3_MEAS.ALARMS.CALIBRATION_MISSING_FIX_4_A AND NOT "DB16000_OPC_UA_TRIGGER_ALARM".CLIENT.U1_STA3_MEAS.ALARMS.CALIBRATION_PROC_A);
   #_w1 := NOT ("M_ONE" AND NOT #ALARM_AUX AND NOT "DB16000_OPC_UA_TRIGGER_ALARM".CLIENT.U1_STA3_MEAS.ALARMS.CALIBRATION_OUT_RANGE_FIX_1_A AND NOT "DB16000_OPC_UA_TRIGGER_ALARM".CLIENT.U1_STA3_MEAS.ALARMS.CALIBRATION_OUT_RANGE_FIX_2_A AND NOT "DB16000_OPC_UA_TRIGGER_ALARM".CLIENT.U1_STA3_MEAS.ALARMS.CALIBRATION_OUT_RANGE_FIX_3_A AND NOT "DB16000_OPC_UA_TRIGGER_ALARM".CLIENT.U1_STA3_MEAS.ALARMS.CALIBRATION_OUT_RANGE_FIX_4_A AND NOT "DB16000_OPC_UA_TRIGGER_ALARM".CLIENT.U1_STA3_MEAS.ALARMS.PLC_PC_MAJOR_VERSIONS_MISMATCH_A);
   IF #_w1 THEN "DB440_MACHINE_ALARM_DECODING".GLOBAL_ALARMS_MACHINE.ALARM_DECODING := 16011; END_IF;
   IF #_w1 AND "M_DUMMY_OFF" THEN
       "DB440_MACHINE_ALARM_DECODING".ALARMS_UNIT_1.ST3_CLADDING.IS_SEOC_ALARMS := TRUE;
   END_IF;
END_REGION

REGION Network 62: SEOC ALARMS
   RUNG wire#powerrail
      Contact( "M_ONE" )
      I_Contact( "DB16000_OPC_UA_TRIGGER_ALARM".CLIENT.U1_STA3_MEAS.ALARMS.MEAS_INITIALIZING_SENSOR_A )
      Not()
      Move(in := 16011, out1 => "DB440_MACHINE_ALARM_DECODING".GLOBAL_ALARMS_MACHINE.ALARM_DECODING)
      Contact( "M_DUMMY_OFF" )
      S_Coil( "DB440_MACHINE_ALARM_DECODING".ALARMS_UNIT_1.ST3_CLADDING.SEOC_ALARMS )
   END_RUNG
   // the same network as SCL:
   #_w1 := NOT ("M_ONE" AND NOT "DB16000_OPC_UA_TRIGGER_ALARM".CLIENT.U1_STA3_MEAS.ALARMS.MEAS_INITIALIZING_SENSOR_A);
   IF #_w1 THEN "DB440_MACHINE_ALARM_DECODING".GLOBAL_ALARMS_MACHINE.ALARM_DECODING := 16011; END_IF;
   IF #_w1 AND "M_DUMMY_OFF" THEN
       "DB440_MACHINE_ALARM_DECODING".ALARMS_UNIT_1.ST3_CLADDING.SEOC_ALARMS := TRUE;
   END_IF;
END_REGION

REGION Network 63: WARNINGS
   RUNG wire#powerrail
      I_Contact( "DB16000_OPC_UA_TRIGGER_ALARM".CLIENT.U1_STA3_MEAS.ALARMS.PLC_PC_MINOR_VERSIONS_MISMATCH_W )
      Not()
      Move(in := #FC_NUMBER, out1 => "DB440_MACHINE_ALARM_DECODING".GLOBAL_ALARMS_MACHINE.WARNING_DECODING)
      wire#w1
      S_Coil( "DB440_MACHINE_ALARM_DECODING".ALARMS_CENTRAL.WARNING )
   END_RUNG
   RUNG wire#w1
      N_Trig( "DB16000_OPC_UA_TRIGGER_ALARM".CLIENT.U1_STA3_MEAS.PULSE.WARNINGS_GONE )
      Move(in := 0, out1 => "DB440_MACHINE_ALARM_DECODING".GLOBAL_ALARMS_MACHINE.WARNING_DECODING)
      R_Coil( "DB440_MACHINE_ALARM_DECODING".ALARMS_CENTRAL.WARNING )
   END_RUNG
   // the same network as SCL:
   #_w1 := NOT (NOT "DB16000_OPC_UA_TRIGGER_ALARM".CLIENT.U1_STA3_MEAS.ALARMS.PLC_PC_MINOR_VERSIONS_MISMATCH_W);
   IF #_w1 THEN
       "DB440_MACHINE_ALARM_DECODING".GLOBAL_ALARMS_MACHINE.WARNING_DECODING := #FC_NUMBER;
       "DB440_MACHINE_ALARM_DECODING".ALARMS_CENTRAL.WARNING := TRUE;
   END_IF;
   #_w2 := NOT #_w1 AND "DB16000_OPC_UA_TRIGGER_ALARM".CLIENT.U1_STA3_MEAS.PULSE.WARNINGS_GONE;   // falling edge
   "DB16000_OPC_UA_TRIGGER_ALARM".CLIENT.U1_STA3_MEAS.PULSE.WARNINGS_GONE := #_w1;
   IF #_w2 THEN
       "DB440_MACHINE_ALARM_DECODING".GLOBAL_ALARMS_MACHINE.WARNING_DECODING := 0;
       "DB440_MACHINE_ALARM_DECODING".ALARMS_CENTRAL.WARNING := FALSE;
   END_IF;
END_REGION
END_FUNCTION
